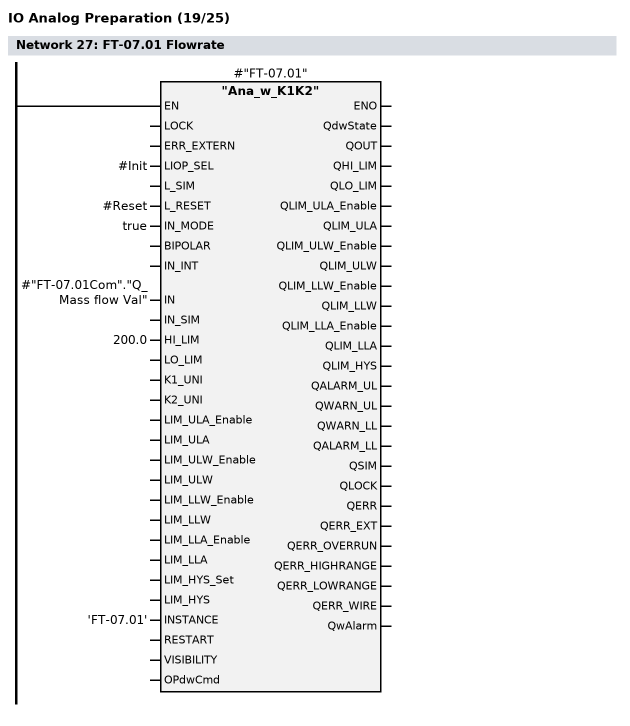
   RUNG wire#powerrail
      #"FT-07.01"(LOCK :=, ERR_EXTERN :=, LIOP_SEL := #Init, L_SIM :=, L_RESET := #Reset, IN_MODE := true, BIPOLAR :=, IN_INT :=, IN := #"FT-07.01Com"."Q_Mass flow Val", IN_SIM :=, HI_LIM := 200.0, LO_LIM :=, K1_UNI :=, K2_UNI :=, LIM_ULA_Enable :=, LIM_ULA :=, LIM_ULW_Enable :=, LIM_ULW :=, LIM_LLW_Enable :=, LIM_LLW :=, LIM_LLA_Enable :=, LIM_LLA :=, LIM_HYS_Set :=, LIM_HYS :=, INSTANCE := 'FT-07.01', RESTART :=, VISIBILITY :=, OPdwCmd :=, QdwState =>, QOUT =>, QHI_LIM =>, QLO_LIM =>, QLIM_ULA_Enable =>, QLIM_ULA =>, QLIM_ULW_Enable =>, QLIM_ULW =>, QLIM_LLW_Enable =>, QLIM_LLW =>, QLIM_LLA_Enable =>, QLIM_LLA =>, QLIM_HYS =>, QALARM_UL =>, QWARN_UL =>, QWARN_LL =>, QALARM_LL =>, QSIM =>, QLOCK =>, QERR =>, QERR_EXT =>, QERR_OVERRUN =>, QERR_HIGHRANGE =>, QERR_LOWRANGE =>, QERR_WIRE =>, QwAlarm =>)
   END_RUNG
   // the same network as SCL:
   #"FT-07.01"(LIOP_SEL := #Init,   // "Ana_w_K1K2"
               L_RESET := #Reset,
               IN_MODE := true,
               IN := #"FT-07.01Com"."Q_Mass flow Val",
               HI_LIM := 200.0,
               INSTANCE := 'FT-07.01');
END_REGION

REGION Network 28: FT-08.01 Communication
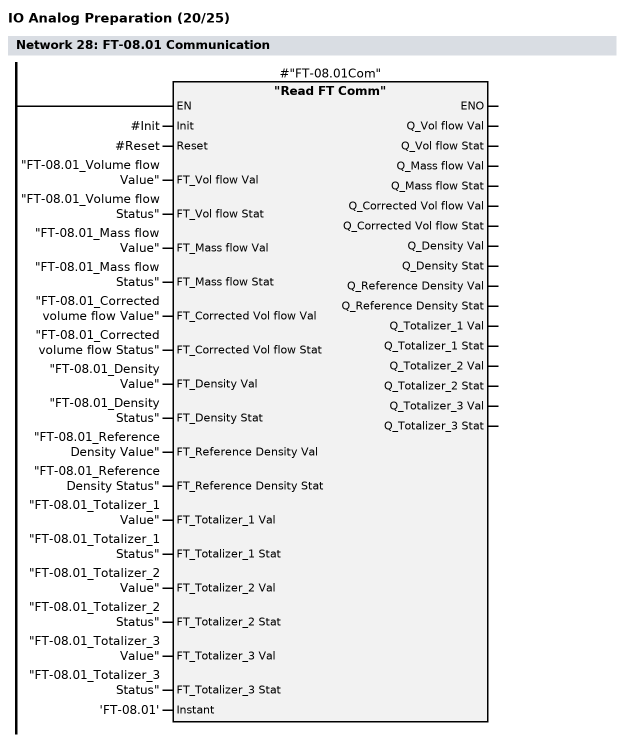
   RUNG wire#powerrail
      #"FT-08.01Com"(Init := #Init, Reset := #Reset, "FT_Vol flow Val" := "FT-08.01_Volume flow Value", "FT_Vol flow Stat" := "FT-08.01_Volume flow Status", "FT_Mass flow Val" := "FT-08.01_Mass flow Value", "FT_Mass flow Stat" := "FT-08.01_Mass flow Status", "FT_Corrected Vol flow Val" := "FT-08.01_Corrected volume flow Value", "FT_Corrected Vol flow Stat" := "FT-08.01_Corrected volume flow Status", "FT_Density Val" := "FT-08.01_Density Value", "FT_Density Stat" := "FT-08.01_Density Status", "FT_Reference Density Val" := "FT-08.01_Reference Density Value", "FT_Reference Density Stat" := "FT-08.01_Reference Density Status", "FT_Totalizer_1 Val" := "FT-08.01_Totalizer_1 Value", "FT_Totalizer_1 Stat" := "FT-08.01_Totalizer_1 Status", "FT_Totalizer_2 Val" := "FT-08.01_Totalizer_2 Value", "FT_Totalizer_2 Stat" := "FT-08.01_Totalizer_2 Status", "FT_Totalizer_3 Val" := "FT-08.01_Totalizer_3 Value", "FT_Totalizer_3 Stat" := "FT-08.01_Totalizer_3 Status", Instant := 'FT-08.01', "Q_Vol flow Val" =>, "Q_Vol flow Stat" =>, "Q_Mass flow Val" =>, "Q_Mass flow Stat" =>, "Q_Corrected Vol flow Val" =>, "Q_Corrected Vol flow Stat" =>, "Q_Density Val" =>, "Q_Density Stat" =>, "Q_Reference Density Val" =>, "Q_Reference Density Stat" =>, "Q_Totalizer_1 Val" =>, "Q_Totalizer_1 Stat" =>, "Q_Totalizer_2 Val" =>, "Q_Totalizer_2 Stat" =>, "Q_Totalizer_3 Val" =>, "Q_Totalizer_3 Stat" =>)
   END_RUNG
   // the same network as SCL:
   #"FT-08.01Com"(Init := #Init,   // "Read FT Comm"
                  Reset := #Reset,
                  "FT_Vol flow Val" := "FT-08.01_Volume flow Value",
                  "FT_Vol flow Stat" := "FT-08.01_Volume flow Status",
                  "FT_Mass flow Val" := "FT-08.01_Mass flow Value",
                  "FT_Mass flow Stat" := "FT-08.01_Mass flow Status",
                  "FT_Corrected Vol flow Val" := "FT-08.01_Corrected volume flow Value",
                  "FT_Corrected Vol flow Stat" := "FT-08.01_Corrected volume flow Status",
                  "FT_Density Val" := "FT-08.01_Density Value",
                  "FT_Density Stat" := "FT-08.01_Density Status",
                  "FT_Reference Density Val" := "FT-08.01_Reference Density Value",
                  "FT_Reference Density Stat" := "FT-08.01_Reference Density Status",
                  "FT_Totalizer_1 Val" := "FT-08.01_Totalizer_1 Value",
                  "FT_Totalizer_1 Stat" := "FT-08.01_Totalizer_1 Status",
                  "FT_Totalizer_2 Val" := "FT-08.01_Totalizer_2 Value",
                  "FT_Totalizer_2 Stat" := "FT-08.01_Totalizer_2 Status",
                  "FT_Totalizer_3 Val" := "FT-08.01_Totalizer_3 Value",
                  "FT_Totalizer_3 Stat" := "FT-08.01_Totalizer_3 Status",
                  Instant := 'FT-08.01');
END_REGION

REGION Network 29: FT-08.01 Flowrate
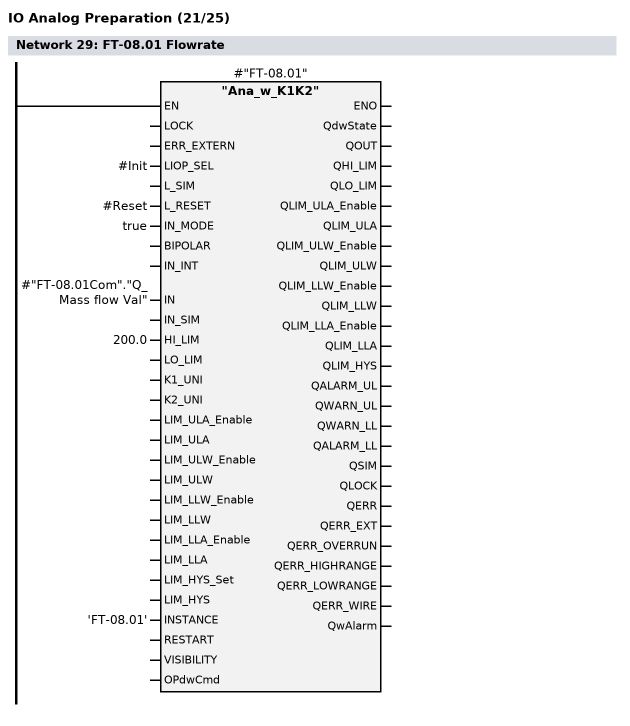
   RUNG wire#powerrail
      #"FT-08.01"(LOCK :=, ERR_EXTERN :=, LIOP_SEL := #Init, L_SIM :=, L_RESET := #Reset, IN_MODE := true, BIPOLAR :=, IN_INT :=, IN := #"FT-08.01Com"."Q_Mass flow Val", IN_SIM :=, HI_LIM := 200.0, LO_LIM :=, K1_UNI :=, K2_UNI :=, LIM_ULA_Enable :=, LIM_ULA :=, LIM_ULW_Enable :=, LIM_ULW :=, LIM_LLW_Enable :=, LIM_LLW :=, LIM_LLA_Enable :=, LIM_LLA :=, LIM_HYS_Set :=, LIM_HYS :=, INSTANCE := 'FT-08.01', RESTART :=, VISIBILITY :=, OPdwCmd :=, QdwState =>, QOUT =>, QHI_LIM =>, QLO_LIM =>, QLIM_ULA_Enable =>, QLIM_ULA =>, QLIM_ULW_Enable =>, QLIM_ULW =>, QLIM_LLW_Enable =>, QLIM_LLW =>, QLIM_LLA_Enable =>, QLIM_LLA =>, QLIM_HYS =>, QALARM_UL =>, QWARN_UL =>, QWARN_LL =>, QALARM_LL =>, QSIM =>, QLOCK =>, QERR =>, QERR_EXT =>, QERR_OVERRUN =>, QERR_HIGHRANGE =>, QERR_LOWRANGE =>, QERR_WIRE =>, QwAlarm =>)
   END_RUNG
   // the same network as SCL:
   #"FT-08.01"(LIOP_SEL := #Init,   // "Ana_w_K1K2"
               L_RESET := #Reset,
               IN_MODE := true,
               IN := #"FT-08.01Com"."Q_Mass flow Val",
               HI_LIM := 200.0,
               INSTANCE := 'FT-08.01');
END_REGION

REGION Network 30: FT-09.01 Communication
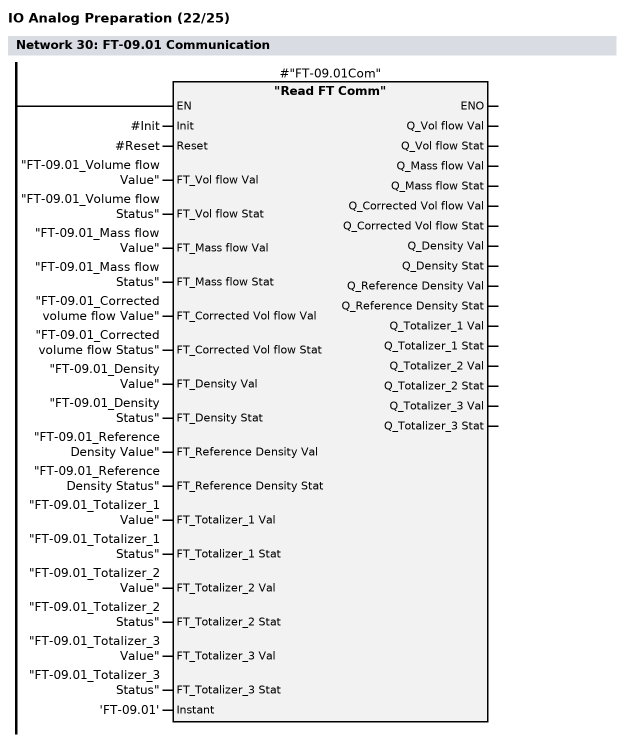
   RUNG wire#powerrail
      #"FT-09.01Com"(Init := #Init, Reset := #Reset, "FT_Vol flow Val" := "FT-09.01_Volume flow Value", "FT_Vol flow Stat" := "FT-09.01_Volume flow Status", "FT_Mass flow Val" := "FT-09.01_Mass flow Value", "FT_Mass flow Stat" := "FT-09.01_Mass flow Status", "FT_Corrected Vol flow Val" := "FT-09.01_Corrected volume flow Value", "FT_Corrected Vol flow Stat" := "FT-09.01_Corrected volume flow Status", "FT_Density Val" := "FT-09.01_Density Value", "FT_Density Stat" := "FT-09.01_Density Status", "FT_Reference Density Val" := "FT-09.01_Reference Density Value", "FT_Reference Density Stat" := "FT-09.01_Reference Density Status", "FT_Totalizer_1 Val" := "FT-09.01_Totalizer_1 Value", "FT_Totalizer_1 Stat" := "FT-09.01_Totalizer_1 Status", "FT_Totalizer_2 Val" := "FT-09.01_Totalizer_2 Value", "FT_Totalizer_2 Stat" := "FT-09.01_Totalizer_2 Status", "FT_Totalizer_3 Val" := "FT-09.01_Totalizer_3 Value", "FT_Totalizer_3 Stat" := "FT-09.01_Totalizer_3 Status", Instant := 'FT-09.01', "Q_Vol flow Val" =>, "Q_Vol flow Stat" =>, "Q_Mass flow Val" =>, "Q_Mass flow Stat" =>, "Q_Corrected Vol flow Val" =>, "Q_Corrected Vol flow Stat" =>, "Q_Density Val" =>, "Q_Density Stat" =>, "Q_Reference Density Val" =>, "Q_Reference Density Stat" =>, "Q_Totalizer_1 Val" =>, "Q_Totalizer_1 Stat" =>, "Q_Totalizer_2 Val" =>, "Q_Totalizer_2 Stat" =>, "Q_Totalizer_3 Val" =>, "Q_Totalizer_3 Stat" =>)
   END_RUNG
   // the same network as SCL:
   #"FT-09.01Com"(Init := #Init,   // "Read FT Comm"
                  Reset := #Reset,
                  "FT_Vol flow Val" := "FT-09.01_Volume flow Value",
                  "FT_Vol flow Stat" := "FT-09.01_Volume flow Status",
                  "FT_Mass flow Val" := "FT-09.01_Mass flow Value",
                  "FT_Mass flow Stat" := "FT-09.01_Mass flow Status",
                  "FT_Corrected Vol flow Val" := "FT-09.01_Corrected volume flow Value",
                  "FT_Corrected Vol flow Stat" := "FT-09.01_Corrected volume flow Status",
                  "FT_Density Val" := "FT-09.01_Density Value",
                  "FT_Density Stat" := "FT-09.01_Density Status",
                  "FT_Reference Density Val" := "FT-09.01_Reference Density Value",
                  "FT_Reference Density Stat" := "FT-09.01_Reference Density Status",
                  "FT_Totalizer_1 Val" := "FT-09.01_Totalizer_1 Value",
                  "FT_Totalizer_1 Stat" := "FT-09.01_Totalizer_1 Status",
                  "FT_Totalizer_2 Val" := "FT-09.01_Totalizer_2 Value",
                  "FT_Totalizer_2 Stat" := "FT-09.01_Totalizer_2 Status",
                  "FT_Totalizer_3 Val" := "FT-09.01_Totalizer_3 Value",
                  "FT_Totalizer_3 Stat" := "FT-09.01_Totalizer_3 Status",
                  Instant := 'FT-09.01');
END_REGION

REGION Network 31: FT-09.01 Flowrate
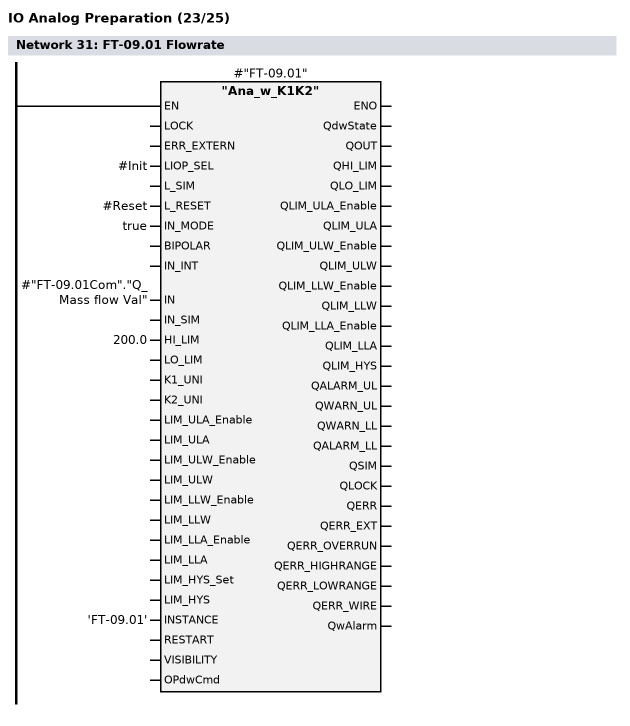
   RUNG wire#powerrail
      #"FT-09.01"(LOCK :=, ERR_EXTERN :=, LIOP_SEL := #Init, L_SIM :=, L_RESET := #Reset, IN_MODE := true, BIPOLAR :=, IN_INT :=, IN := #"FT-09.01Com"."Q_Mass flow Val", IN_SIM :=, HI_LIM := 200.0, LO_LIM :=, K1_UNI :=, K2_UNI :=, LIM_ULA_Enable :=, LIM_ULA :=, LIM_ULW_Enable :=, LIM_ULW :=, LIM_LLW_Enable :=, LIM_LLW :=, LIM_LLA_Enable :=, LIM_LLA :=, LIM_HYS_Set :=, LIM_HYS :=, INSTANCE := 'FT-09.01', RESTART :=, VISIBILITY :=, OPdwCmd :=, QdwState =>, QOUT =>, QHI_LIM =>, QLO_LIM =>, QLIM_ULA_Enable =>, QLIM_ULA =>, QLIM_ULW_Enable =>, QLIM_ULW =>, QLIM_LLW_Enable =>, QLIM_LLW =>, QLIM_LLA_Enable =>, QLIM_LLA =>, QLIM_HYS =>, QALARM_UL =>, QWARN_UL =>, QWARN_LL =>, QALARM_LL =>, QSIM =>, QLOCK =>, QERR =>, QERR_EXT =>, QERR_OVERRUN =>, QERR_HIGHRANGE =>, QERR_LOWRANGE =>, QERR_WIRE =>, QwAlarm =>)
   END_RUNG
   // the same network as SCL:
   #"FT-09.01"(LIOP_SEL := #Init,   // "Ana_w_K1K2"
               L_RESET := #Reset,
               IN_MODE := true,
               IN := #"FT-09.01Com"."Q_Mass flow Val",
               HI_LIM := 200.0,
               INSTANCE := 'FT-09.01');
END_REGION

REGION Network 32: FT-10.01 Communication
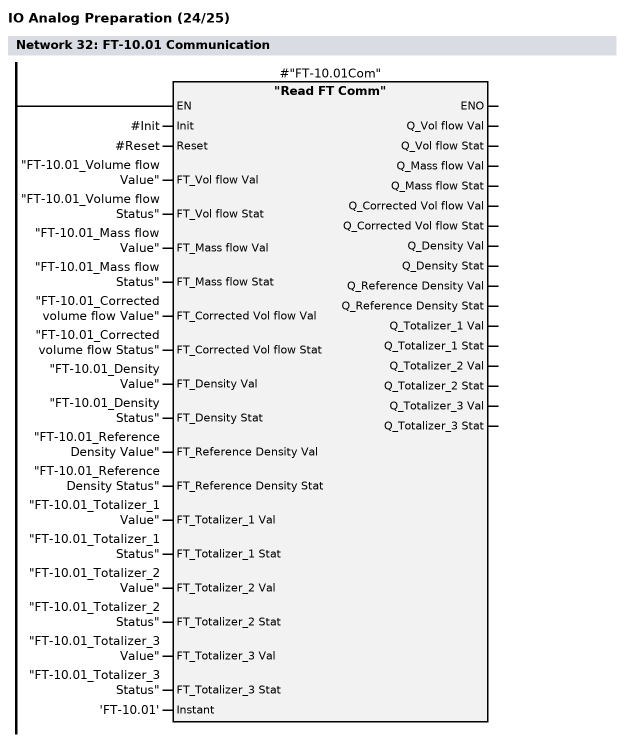
   RUNG wire#powerrail
      #"FT-10.01Com"(Init := #Init, Reset := #Reset, "FT_Vol flow Val" := "FT-10.01_Volume flow Value", "FT_Vol flow Stat" := "FT-10.01_Volume flow Status", "FT_Mass flow Val" := "FT-10.01_Mass flow Value", "FT_Mass flow Stat" := "FT-10.01_Mass flow Status", "FT_Corrected Vol flow Val" := "FT-10.01_Corrected volume flow Value", "FT_Corrected Vol flow Stat" := "FT-10.01_Corrected volume flow Status", "FT_Density Val" := "FT-10.01_Density Value", "FT_Density Stat" := "FT-10.01_Density Status", "FT_Reference Density Val" := "FT-10.01_Reference Density Value", "FT_Reference Density Stat" := "FT-10.01_Reference Density Status", "FT_Totalizer_1 Val" := "FT-10.01_Totalizer_1 Value", "FT_Totalizer_1 Stat" := "FT-10.01_Totalizer_1 Status", "FT_Totalizer_2 Val" := "FT-10.01_Totalizer_2 Value", "FT_Totalizer_2 Stat" := "FT-10.01_Totalizer_2 Status", "FT_Totalizer_3 Val" := "FT-10.01_Totalizer_3 Value", "FT_Totalizer_3 Stat" := "FT-10.01_Totalizer_3 Status", Instant := 'FT-10.01', "Q_Vol flow Val" =>, "Q_Vol flow Stat" =>, "Q_Mass flow Val" =>, "Q_Mass flow Stat" =>, "Q_Corrected Vol flow Val" =>, "Q_Corrected Vol flow Stat" =>, "Q_Density Val" =>, "Q_Density Stat" =>, "Q_Reference Density Val" =>, "Q_Reference Density Stat" =>, "Q_Totalizer_1 Val" =>, "Q_Totalizer_1 Stat" =>, "Q_Totalizer_2 Val" =>, "Q_Totalizer_2 Stat" =>, "Q_Totalizer_3 Val" =>, "Q_Totalizer_3 Stat" =>)
   END_RUNG
   // the same network as SCL:
   #"FT-10.01Com"(Init := #Init,   // "Read FT Comm"
                  Reset := #Reset,
                  "FT_Vol flow Val" := "FT-10.01_Volume flow Value",
                  "FT_Vol flow Stat" := "FT-10.01_Volume flow Status",
                  "FT_Mass flow Val" := "FT-10.01_Mass flow Value",
                  "FT_Mass flow Stat" := "FT-10.01_Mass flow Status",
                  "FT_Corrected Vol flow Val" := "FT-10.01_Corrected volume flow Value",
                  "FT_Corrected Vol flow Stat" := "FT-10.01_Corrected volume flow Status",
                  "FT_Density Val" := "FT-10.01_Density Value",
                  "FT_Density Stat" := "FT-10.01_Density Status",
                  "FT_Reference Density Val" := "FT-10.01_Reference Density Value",
                  "FT_Reference Density Stat" := "FT-10.01_Reference Density Status",
                  "FT_Totalizer_1 Val" := "FT-10.01_Totalizer_1 Value",
                  "FT_Totalizer_1 Stat" := "FT-10.01_Totalizer_1 Status",
                  "FT_Totalizer_2 Val" := "FT-10.01_Totalizer_2 Value",
                  "FT_Totalizer_2 Stat" := "FT-10.01_Totalizer_2 Status",
                  "FT_Totalizer_3 Val" := "FT-10.01_Totalizer_3 Value",
                  "FT_Totalizer_3 Stat" := "FT-10.01_Totalizer_3 Status",
                  Instant := 'FT-10.01');
END_REGION

REGION Network 33: FT-10.01 Flowrate
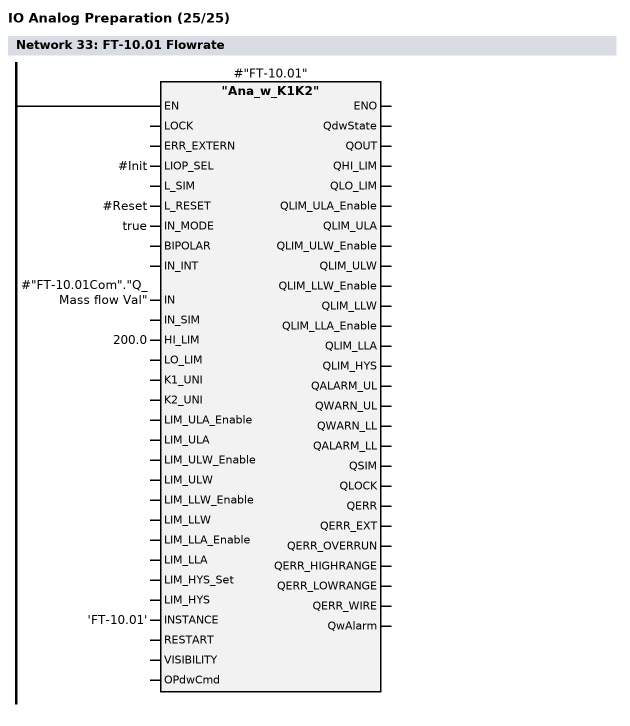
   RUNG wire#powerrail
      #"FT-10.01"(LOCK :=, ERR_EXTERN :=, LIOP_SEL := #Init, L_SIM :=, L_RESET := #Reset, IN_MODE := true, BIPOLAR :=, IN_INT :=, IN := #"FT-10.01Com"."Q_Mass flow Val", IN_SIM :=, HI_LIM := 200.0, LO_LIM :=, K1_UNI :=, K2_UNI :=, LIM_ULA_Enable :=, LIM_ULA :=, LIM_ULW_Enable :=, LIM_ULW :=, LIM_LLW_Enable :=, LIM_LLW :=, LIM_LLA_Enable :=, LIM_LLA :=, LIM_HYS_Set :=, LIM_HYS :=, INSTANCE := 'FT-10.01', RESTART :=, VISIBILITY :=, OPdwCmd :=, QdwState =>, QOUT =>, QHI_LIM =>, QLO_LIM =>, QLIM_ULA_Enable =>, QLIM_ULA =>, QLIM_ULW_Enable =>, QLIM_ULW =>, QLIM_LLW_Enable =>, QLIM_LLW =>, QLIM_LLA_Enable =>, QLIM_LLA =>, QLIM_HYS =>, QALARM_UL =>, QWARN_UL =>, QWARN_LL =>, QALARM_LL =>, QSIM =>, QLOCK =>, QERR =>, QERR_EXT =>, QERR_OVERRUN =>, QERR_HIGHRANGE =>, QERR_LOWRANGE =>, QERR_WIRE =>, QwAlarm =>)
   END_RUNG
   // the same network as SCL:
   #"FT-10.01"(LIOP_SEL := #Init,   // "Ana_w_K1K2"
               L_RESET := #Reset,
               IN_MODE := true,
               IN := #"FT-10.01Com"."Q_Mass flow Val",
               HI_LIM := 200.0,
               INSTANCE := 'FT-10.01');
END_REGION
END_FUNCTION_BLOCK

FUNCTION_BLOCK "Ana_w_K1K2"
TITLE = Analogue
{ S7_Optimized_Access := 'FALSE' }
AUTHOR : RM
FAMILY : MON
VERSION : 0.1
   VAR_INPUT 
      LOCK : Bool;
      ERR_EXTERN : Bool;
      LIOP_SEL : Bool;
      L_SIM : Bool;
      L_RESET : Bool;
      IN_MODE : Bool;
      BIPOLAR : Bool;
      IN_INT : Int := 0;
      IN : Real := 55.0;
      IN_SIM : Real := 55.0;
      HI_LIM : Real := 100.0;
      LO_LIM : Real;
      K1_UNI : Real;   // Low Measuring Unit
      K2_UNI : Real := 27648.0;   // High Mesuring Unit
      LIM_ULA_Enable : Bool;
      LIM_ULA : Real := 90.0;
      LIM_ULW_Enable : Bool;
      LIM_ULW : Real := 80.0;
      LIM_LLW_Enable : Bool;
      LIM_LLW : Real := 20.0;
      LIM_LLA_Enable : Bool;
      LIM_LLA : Real := 10.0;
      LIM_HYS_Set : Bool;
      LIM_HYS : Real;
      INSTANCE : String := 'Analogue_001';
      RESTART : Bool;
   END_VAR

   VAR_OUTPUT 
      QdwState : DWord;
      QOUT : Real;
      QHI_LIM : Real;
      QLO_LIM : Real;
      QLIM_ULA_Enable : Bool;
      QLIM_ULA : Real;
      QLIM_ULW_Enable : Bool;
      QLIM_ULW : Real;
      QLIM_LLW_Enable : Bool;
      QLIM_LLW : Real;
      QLIM_LLA_Enable : Bool;
      QLIM_LLA : Real;
      QLIM_HYS : Real;
      QALARM_UL : Bool;
      QWARN_UL : Bool;
      QWARN_LL : Bool;
      QALARM_LL : Bool;
      QSIM : Bool;
      QLOCK : Bool;
      QERR : Bool;
      QERR_EXT : Bool;
      QERR_OVERRUN : Bool;
      QERR_HIGHRANGE : Bool;
      QERR_LOWRANGE : Bool;
      QERR_WIRE : Bool;
      QwAlarm : Word;
   END_VAR

   VAR_IN_OUT 
      VISIBILITY : Byte := 0;
      OPdwCmd : DWord;
   END_VAR

   VAR 
      OP_RESET : Bool;
      QLIM_HYS_Set : Bool;
      QIN_MODE : Bool;
      OP_LIM_ULA : Real;
      OP_LIM_ULW : Real;
      OP_LIM_LLW : Real;
      OP_LIM_LLA : Real;
      OP_SIM_Value : Real;
      OP_LIM_HYS_Perc : Real;
      OP_LIM_HYS_Abs : Real;
      OP_HI_LIM : Real;
      OP_LO_LIM : Real;
      OP_VISIBILITY : Byte;
      VISIBILITY_OLD : Byte;
      SEF_L_RESET_Link : Bool;
      Condition_SEF_L_RESET_Link : Bool;
      SEF_L_RESET_OP : Bool;
      Condition_Enable_ULA : Bool;
      Condition_Enable_ULW : Bool;
      Condition_Enable_LLW : Bool;
      Condition_Enable_LLA : Bool;
   END_VAR


BEGIN
	(*
	Network 1: Start up
	*)
	IF #RESTART= true THEN
	  #QOUT:= 0;
	  #OPdwCmd:=0;
	END_IF;
	
	(*
	Network 2: Simulation On/Off
	Vaiable: OPdwCmd  Bit:  20  =  Process
	Vaiable: OPdwCmd  Bit:  21  =  Simulation
	*)
	IF (#LIOP_SEL=true AND #L_SIM=true) OR (#OPdwCmd.%X21=true AND #LIOP_SEL=false) THEN
	  #QSIM:=true;
	  #OPdwCmd.%X20:=false;
	  #OPdwCmd.%X21:=false;
	ELSIF (#LIOP_SEL=true AND #L_SIM=false) OR (#OPdwCmd.%X20=true AND #LIOP_SEL=false) THEN
	  #QSIM:= false;
	  #OPdwCmd.%X20:=false;
	  #OPdwCmd.%X21:=false;
	END_IF;
	
	(*
	Network 3: Mode limit Hysteresis
	Vaiable: OPdwCmd  Bit:  12  =  Hysteresis Percental
	Vaiable: OPdwCmd  Bit:  13  =  Hysteresis Absolute
	*)
	IF (#LIOP_SEL=true AND #LIM_HYS_Set=true) OR (#OPdwCmd.%X13=true AND #LIOP_SEL=false) THEN
	  #QLIM_HYS_Set:=true;
	  #OPdwCmd.%X12:=false;
	  #OPdwCmd.%X13:=false;
	ELSIF (#LIOP_SEL=true AND #LIM_HYS_Set=false) OR (#OPdwCmd.%X12=true AND #LIOP_SEL=false) THEN
	  #QLIM_HYS_Set:=false;
	  #OPdwCmd.%X12:=false;
	  #OPdwCmd.%X13:=false;
	END_IF;
	
	(*
	Network 4: Mode Periphery / Real value
	Vaiable: OPdwCmd  Bit:  14  =  Periphery
	Vaiable: OPdwCmd  Bit:  15  =  Real value
	*)
	IF (#LIOP_SEL=true AND #IN_MODE=true) OR (#OPdwCmd.%X15=true AND #LIOP_SEL=false) THEN
	  #QIN_MODE:=true;
	  #OPdwCmd.%X14:=false;
	  #OPdwCmd.%X15:=false;
	ELSIF (#LIOP_SEL=true AND #IN_MODE=false) OR (#OPdwCmd.%X14=true AND #LIOP_SEL=false) THEN
	  #QIN_MODE:=false;
	  #OPdwCmd.%X14:=false;
	  #OPdwCmd.%X15:=false;
	END_IF;
	
	(*
	Network 5: Reset Operation
	Vaiable: OPdwCmd  Bit:  24  =  Reset
	*)
	// Rising edge by linking
	IF #L_RESET=true AND #Condition_SEF_L_RESET_Link=false THEN
	  #SEF_L_RESET_Link:=true;
	  #Condition_SEF_L_RESET_Link:=true;
	ELSIF #L_RESET=true AND #Condition_SEF_L_RESET_Link=true THEN
	  #SEF_L_RESET_Link:=false;
	ELSE
	  #Condition_SEF_L_RESET_Link:=false;
	END_IF;
	// Rising edge by operator
	IF #OPdwCmd.%X24=true THEN
	  #SEF_L_RESET_OP:=true;
	  #OPdwCmd.%X24:=false;
	ELSE
	  #SEF_L_RESET_OP:=false;
	END_IF;
	// Reset error #OP_RESET:=(#LIOP_SEL=true AND #SEF_L_RESET_Link=true) OR (#SEF_L_RESET_OP=true AND #LIOP_SEL=false);
	#OP_RESET:=(#L_RESET=true) OR (#SEF_L_RESET_OP=true AND #LIOP_SEL=false);
	
	(*
	Network 6: Enable alarm for upper limit
	Vaiable: OPdwCmd  Bit:  0  =  Enable alarm upper limit
	*)
	IF #OPdwCmd.%X0=true THEN
	  #Condition_Enable_ULA:=NOT #Condition_Enable_ULA;
	  #OPdwCmd.%X0:=false;
	END_IF;
	//IF (#LIOP_SEL=true AND #LIM_ULA_Enable=true) OR (#LIOP_SEL=false AND #Condition_Enable_ULA=true) THEN  
	//#QLIM_ULA_Enable := true;
	//ELSIF (#LIOP_SEL=true AND #LIM_ULA_Enable=false) OR (#LIOP_SEL=false AND #Condition_Enable_ULA=false) THEN
	//    #QLIM_ULA_Enable := false;
	//END_IF;
	IF ( #LIM_ULA_Enable=true) OR (#LIOP_SEL=false AND #Condition_Enable_ULA=true) THEN  
	  #QLIM_ULA_Enable:=true;
	ELSIF (#LIOP_SEL=true AND #LIM_ULA_Enable=false) OR (#LIOP_SEL=false AND #Condition_Enable_ULA=false) THEN
	  #QLIM_ULA_Enable:=false;
	END_IF;
	
	  
	(*
	Network 7: Enable warning for upper limit
	Vaiable: OPdwCmd  Bit:  1  =  Enable warning upper limit
	*)
	IF #OPdwCmd.%X1=true THEN
	  #Condition_Enable_ULW:=NOT #Condition_Enable_ULW;
	  #OPdwCmd.%X1:=false;
	END_IF;
	
	IF ( #LIM_ULW_Enable=true) OR (#LIOP_SEL=false AND #Condition_Enable_ULW=true) THEN  
	  #QLIM_ULW_Enable:=true;
	ELSIF (#LIOP_SEL=true AND #LIM_ULW_Enable=false) OR (#LIOP_SEL=false AND #Condition_Enable_ULW=false) THEN
	  #QLIM_ULW_Enable:=false;
	END_IF;
	
	(*
	Network 8: Enable warning for lower limit
	Vaiable: OPdwCmd  Bit:  2  =  Enable warning lower limit
	*)
	IF #OPdwCmd.%X2=true THEN
	  #Condition_Enable_LLW:=NOT #Condition_Enable_LLW ;
	  #OPdwCmd.%X2:=false;
	END_IF;
	
	IF ( #LIM_LLW_Enable=true) OR (#LIOP_SEL=false AND #Condition_Enable_LLW=true) THEN  
	  #QLIM_LLW_Enable:=true;
	ELSIF (#LIOP_SEL=true AND #LIM_LLW_Enable=false) OR (#LIOP_SEL=false AND #Condition_Enable_LLW=false) THEN
	  #QLIM_LLW_Enable:=false;
	END_IF;
	
	(*
	Network 9: Enable alarm for lower limit
	Vaiable: OPdwCmd  Bit:  3  =  Enable alarm lower limit
	*)
	IF #OPdwCmd.%X3=true THEN
	  #Condition_Enable_LLA:=NOT #Condition_Enable_LLA;
	  #OPdwCmd.%X3:=false;
	END_IF;
	
	IF ( #LIM_LLA_Enable=true) OR (#LIOP_SEL=false AND #Condition_Enable_LLA=true) THEN  
	  #QLIM_LLA_Enable:=true;
	ELSIF (#LIOP_SEL=true AND #LIM_LLA_Enable=false) OR (#LIOP_SEL=false AND #Condition_Enable_LLA=false) THEN
	  #QLIM_LLA_Enable:=false;
	END_IF;
	
	(*
	Network 10: Calculate hysteresis value
	*)
	IF #LIOP_SEL=true AND #QLIM_HYS_Set=true THEN
	  // Absolute by PLC
	  #OP_HI_LIM:=#HI_LIM;
	  #OP_LO_LIM:=#LO_LIM;
	  #OP_LIM_HYS_Perc:=#LIM_HYS/((#HI_LIM-#LO_LIM)/100);
	  #OP_LIM_HYS_Abs:=#LIM_HYS;
	  #QHI_LIM:=#HI_LIM;
	  #QLO_LIM:=#LO_LIM;
	  #QLIM_HYS:=#OP_LIM_HYS_Abs;
	ELSIF #LIOP_SEL=true AND #QLIM_HYS_Set=false THEN
	  // Percental by PLC
	  #OP_HI_LIM:=#HI_LIM;
	  #OP_LO_LIM:=#LO_LIM;
	  #OP_LIM_HYS_Perc:=#LIM_HYS;
	  #OP_LIM_HYS_Abs:=#LIM_HYS*((#HI_LIM-#LO_LIM)/100);
	  #QHI_LIM:=#HI_LIM;
	  #QLO_LIM:=#LO_LIM;
	  #QLIM_HYS:=#OP_LIM_HYS_Abs;
	ELSIF #LIOP_SEL=false AND #QLIM_HYS_Set=true THEN
	  // Absolute by operator
	  #QHI_LIM:=#OP_HI_LIM;
	  #QLO_LIM:=#OP_LO_LIM;
	  #OP_LIM_HYS_Perc:=#OP_LIM_HYS_Abs/((#OP_HI_LIM-#OP_LO_LIM)/100);
	  #QLIM_HYS:=#OP_LIM_HYS_Abs;
	ELSE
	  // Percental by operator
	  #QHI_LIM:=#OP_HI_LIM;
	  #QLO_LIM:=#OP_LO_LIM;
	  #OP_LIM_HYS_Abs:=#OP_LIM_HYS_Perc*((#OP_HI_LIM-#OP_LO_LIM)/100);
	  #QLIM_HYS:=#OP_LIM_HYS_Abs;
	END_IF;
	
	//Transfer output to simulation value in process mode
	IF #QSIM=false THEN
	  #IN_SIM:=#QOUT;
	END_IF;
	(*
	Network 11: Convert integer to real and scale it to selcted mode
	*)
	IF #QIN_MODE=false AND #QSIM=false AND #BIPOLAR=false THEN
	  // Convert integer to real and scale in unipolar mode (4..20mA)
	    #QOUT:=(((INT_TO_REAL(#IN_INT)-#K1_UNI)/#K2_UNI)*(#HI_LIM-#LO_LIM))+#LO_LIM;
	ELSIF #QIN_MODE=false AND #QSIM=false AND #BIPOLAR=true THEN
	  // Convert integer to real and scale in bipolar mode (4..20mA)
	  #QOUT:=(((INT_TO_REAL(#IN_INT)+27648)/55296)*(#HI_LIM-#LO_LIM))+#LO_LIM;
	END_IF;
	
	//Che errors
	#QERR_EXT:=#ERR_EXTERN;
	#QLOCK:=#LOCK;
	
	(*
	Network 12: Check errors for simulation mode or real value
	*)
	IF (#QIN_MODE=true OR #QSIM=true) AND #QHI_LIM>=#QOUT AND #QLO_LIM<=#QOUT THEN
	    #QERR_OVERRUN:=false;
	    #QERR_HIGHRANGE:=false;
	    #QERR_LOWRANGE:=false;
	    #QERR_WIRE:=false;
	  END_IF;
	
	(*
	Network 13: Check errors for periphery unipolar mode (4..20mA)
	*)
	(*
	    Measuring Range   Units       Range
	    (4..20mA)         (Dez)
	    ============================================
	    >22,81            >32511      Overrun
	    --------------------------------------------
	    22,81              32511
	      .                           High range
	    20,01              27649         
	    --------------------------------------------
	    20,00              27648 
	      .                           Nominal range
	     4,00                  0
	    --------------------------------------------
	     3,99                 -1
	      .                           Low range
	     1,185             -4864
	    --------------------------------------------
	    <1,185            <-4864      Wire breakage
	*)
	IF #QSIM=false AND #QIN_MODE=false AND #BIPOLAR=false THEN
	  CASE #IN_INT OF
	      -4864..-1 :      // Low range
	    #QERR_OVERRUN:=false;
	    #QERR_HIGHRANGE:=false;
	   // #QERR_LOWRANGE := true;
	    #QERR_WIRE:=false;
	    0.. 27648:       // Nominal range
	    #QERR_OVERRUN:=false;
	    #QERR_HIGHRANGE:=false;
	    #QERR_LOWRANGE:=false;
	    #QERR_WIRE:=false;
	    27649..32511:   // High range
	    #QERR_OVERRUN:=false;
	    #QERR_HIGHRANGE:=true;
	    #QERR_LOWRANGE := false;
	    #QERR_WIRE:=false;
	  ELSE
	    IF #IN_INT>32511 THEN
	      // Overrun
	      #QERR_OVERRUN:=true;
	      #QERR_HIGHRANGE:=false;
	      #QERR_LOWRANGE:=false;
	      #QERR_WIRE:=false;
	    ELSE
	      // Wire breakage
	      #QERR_OVERRUN:=false;
	      #QERR_HIGHRANGE:=false;
	      #QERR_LOWRANGE:=false;
	      #QERR_WIRE:=true;
	    END_IF;  
	  END_CASE;
	END_IF;
	
	(*
	Network 14: Check errors for periphery bipolar mode (4..20mA)
	*)
	(*
	    Measuring Range   Units       Range
	    (4..20mA)         (Dez)
	    ============================================
	    >22,81            >32511      Overrun
	    --------------------------------------------
	    22,81              32511
	      .                           High range
	    20,01              27649         
	    --------------------------------------------
	    20,00              27648 
	      .                           Nominal range
	     4,00             -27648
	    --------------------------------------------
	     3,99             -27649
	      .                           Low range
	     1,185            -32512
	    --------------------------------------------
	    <1,185           <-32512      Wire breakage
	*)
	IF #QSIM=false AND #QIN_MODE=false AND #BIPOLAR=true THEN
	  CASE #IN_INT OF
	    -32512..-27649:         // Low range
	    #QERR_OVERRUN:=false;
	    #QERR_HIGHRANGE:=false;
	    #QERR_LOWRANGE:=true;
	    #QERR_WIRE:=false;
	    -27648..27648:         // Nominal range
	    #QERR_OVERRUN:=false;
	    #QERR_HIGHRANGE:=false;
	    #QERR_LOWRANGE:=false;
	    #QERR_WIRE:=false;
	    27649..32511:         // High range
	    #QERR_OVERRUN:=false;
	    #QERR_HIGHRANGE:=true;
	    #QERR_LOWRANGE:=false;
	    #QERR_WIRE:=false;
	  ELSE
	    IF #IN_INT>32511 THEN
	      // Overrun
	      #QERR_OVERRUN:=true;
	      #QERR_HIGHRANGE:=false;
	      #QERR_LOWRANGE:=false;
	      #QERR_WIRE:=false;
	    ELSE
	      // Wire breakage
	      #QERR_OVERRUN:=false;
	      #QERR_HIGHRANGE:=false;
	      #QERR_LOWRANGE:=false;
	      #QERR_WIRE:=true;
	    END_IF;  
	  END_CASE;
	END_IF;
	
	(*
	Network 15: Check range error for real value
	*)
	//  Check for high range injury
	IF (#IN>#QHI_LIM AND #QIN_MODE=true AND #QSIM=false AND #LIOP_SEL=true) OR
	   (#IN_SIM>#QHI_LIM AND #QSIM=true AND #LIOP_SEL=true) OR
	   (#OP_SIM_Value>#QHI_LIM AND #QSIM=true AND #LIOP_SEL=false) THEN
	      #QERR_HIGHRANGE:=true;
	END_IF;
	//  Check for low range injury
	IF (#IN<#QLO_LIM AND #QIN_MODE=true AND #QSIM=false AND #LIOP_SEL=true) OR
	   (#IN_SIM<#QLO_LIM AND #QSIM=true AND #LIOP_SEL=true) OR
	   (#OP_SIM_Value<#QLO_LIM AND #QSIM=true AND #LIOP_SEL=false) THEN
	      #QERR_LOWRANGE:=true;
	END_IF;
	    
	(*
	Network 16: General Error
	*)
	IF #OP_RESET=true THEN
	  #QERR:=false;
	ELSIF #QERR_EXT=true OR #QLOCK=true OR #QERR_OVERRUN OR #QERR_WIRE THEN
	  #QERR:=true;
	END_IF;
	
	(*
	Network 17: Upper limit alarm
	*)
	IF #QLIM_ULA_Enable=true THEN
	  IF #QLIM_ULA<=#QOUT THEN
	    #QALARM_UL:=true;
	  ELSIF (#QLIM_ULA-#QLIM_HYS)>#QOUT THEN
	    #QALARM_UL:=false;
	  END_IF;
	ELSE
	  #QALARM_UL:=false;
	END_IF;
	 
	(*
	Network 18: Upper limit warning
	*)
	IF #QLIM_ULW_Enable=true THEN
	  IF #QLIM_ULW<=#QOUT THEN
	    #QWARN_UL:=true;
	  ELSIF (#QLIM_ULW-#QLIM_HYS)>#QOUT THEN
	    #QWARN_UL:=false;
	  END_IF;
	ELSE
	  #QWARN_UL:=false;
	END_IF;
	
	(*
	Network 19: Lower limit warning
	*)
	IF #QLIM_LLW_Enable=true THEN
	  IF #QLIM_LLW>=#QOUT THEN
	    #QWARN_LL:=true;
	  ELSIF (#QLIM_LLW+#QLIM_HYS)<#QOUT THEN
	    #QWARN_LL:=false;
	  END_IF;
	ELSE
	  #QWARN_LL:=false;
	END_IF;
	
	(*
	Network 20: Lower limit alarm
	*)
	IF #QLIM_LLA_Enable=true THEN
	  IF #QLIM_LLA>=#QOUT THEN
	    #QALARM_LL:=true;
	  ELSIF (#QLIM_LLA+#QLIM_HYS)<#QOUT THEN
	    #QALARM_LL:=false;
	  END_IF;
	ELSE
	  #QALARM_LL:=false;
	END_IF;
	
	(*
	Network 21: Set limit value
	*)
	IF #QSIM=true AND #LIOP_SEL=false THEN
	  // Set values in simulation mode by operator
	  #QHI_LIM:=#OP_HI_LIM;
	  #QLO_LIM:=#OP_LO_LIM;
	  #QLIM_ULA:=#OP_LIM_ULA;
	  #QLIM_ULW:=#OP_LIM_ULW;
	  #QLIM_LLW:=#OP_LIM_LLW;
	  #QLIM_LLA:=#OP_LIM_LLA;
	ELSE
	  // Set values in normal mode by linking
	  #OP_HI_LIM:=#HI_LIM;
	  #QHI_LIM:=#HI_LIM;
	  #OP_LO_LIM:=#LO_LIM;
	  #QLO_LIM:=#LO_LIM;
	  #OP_LIM_ULA:=#LIM_ULA;
	  #QLIM_ULA:=#LIM_ULA;
	  #OP_LIM_ULW:=#LIM_ULW;
	  #QLIM_ULW:=#LIM_ULW;
	  #OP_LIM_LLW:=#LIM_LLW;
	  #QLIM_LLW:=#LIM_LLW;
	  #OP_LIM_LLA:=#LIM_LLA;
	  #QLIM_LLA:=#LIM_LLA;
	END_IF;
	
	(*
	Network 22: Check settings and values
	*)
	IF #QSIM=false AND #QIN_MODE=true THEN
	  // Set settings in process mode by PLC (real value)
	  #QOUT:=#IN;
	ELSIF #QSIM=true AND #LIOP_SEL=false THEN
	  // Set settings in simulation mode by operator (real value)
	  #QOUT:=#OP_SIM_Value;
	ELSIF #QSIM=true AND #LIOP_SEL=true THEN
	  // Set settings in simulation mode by PLC (real value)
	  #QOUT:=#IN_SIM;
	END_IF;
	
	IF #QSIM=false AND #LIOP_SEL=true AND #IN_MODE=false THEN
	  //Set settings in process mode by PLC (periphery)
	  IF #QERR_EXT=true OR #QLOCK=true THEN
	  //Set value in case of error
	    #QOUT:=#QLO_LIM;
	ELSE
	  IF #QOUT>#QHI_LIM THEN
	    #QOUT:=#QHI_LIM;
	  ELSIF #QOUT<#LO_LIM THEN
	    #QOUT:=#QLO_LIM;
	  END_IF;
	END_IF;
	END_IF;
	(*
	Network 23: Infuence visibility of faceplate window
	*)
	IF #OP_VISIBILITY<>#VISIBILITY_OLD THEN
	  #VISIBILITY_OLD:=#OP_VISIBILITY;
	  #VISIBILITY:=#OP_VISIBILITY;
	ELSIF #VISIBILITY<>#VISIBILITY_OLD THEN
	  #VISIBILITY_OLD:=#VISIBILITY;
	  #OP_VISIBILITY:=#VISIBILITY;
	END_IF;
	
	(*
	Network 24: Transfer output to simulation value in process mode
	*)
	IF #QSIM=false THEN
	  #IN_SIM:=#QOUT;
	END_IF;
	
	(*
	Network 25: Check errors
	*)
	#QERR_EXT:=#ERR_EXTERN;
	#QLOCK:=#LOCK;
	
	(*
	Network 26: Set state for HMI
	*)
	#QdwState.%X0:= #QIN_MODE;
	#QdwState.%X1:=#QLIM_HYS_Set;
	#QdwState.%X2:=false;
	#QdwState.%X3:=false;
	#QdwState.%X4:=#QLIM_ULA_Enable;
	#QdwState.%X5:=#QLIM_ULW_Enable;
	#QdwState.%X6:=#QLIM_LLW_Enable;
	#QdwState.%X7:=#QLIM_LLA_Enable;
	#QdwState.%X9:=#QALARM_LL OR #QALARM_UL;
	#QdwState.%X8:=NOT #QdwState.%X9 AND (#QWARN_LL OR #QWARN_UL);
	#QdwState.%X10:=false;
	#QdwState.%X11:=false;
	#QdwState.%X12:=#QERR_LOWRANGE;
	#QdwState.%X13:=#QERR_HIGHRANGE;
	#QdwState.%X14:=#QERR_OVERRUN;
	#QdwState.%X15:=#QERR_WIRE;
	#QdwState.%X16:=false;
	#QdwState.%X17:=false;
	#QdwState.%X18:=#QSIM;
	#QdwState.%X19:=false;
	#QdwState.%X20:=false;
	#QdwState.%X21:=false;
	#QdwState.%X22:=false;
	#QdwState.%X23:=false;
	#QdwState.%X24:=#QERR;
	#QdwState.%X25:=#QERR_EXT;
	#QdwState.%X26:=#QLOCK;
	#QdwState.%X27:=#LOCK;
	#QdwState.%X28:=false;
	#QdwState.%X29:=false;
	#QdwState.%X30:=false;
	#QdwState.%X31:=false;
	
	(*
	Network 27: Bit alarm procedure
	*)
	#QwAlarm.%X0:=#QALARM_LL;
	#QwAlarm.%X1:=#QALARM_UL;
	#QwAlarm.%X2:=false;
	#QwAlarm.%X3:=false;
	#QwAlarm.%X4:=#QLOCK;
	#QwAlarm.%X5:=false;
	#QwAlarm.%X6:=#QERR_EXT;
	#QwAlarm.%X7:=#QERR;
	#QwAlarm.%X8:=#QWARN_LL;
	#QwAlarm.%X9:=#QWARN_UL;
	#QwAlarm.%X10:=false;
	#QwAlarm.%X11:=false;
	#QwAlarm.%X12:=#LOCK;
	#QwAlarm.%X13:=false;
	#QwAlarm.%X14:=false;
	#QwAlarm.%X15:=#QSIM;
	
END_FUNCTION_BLOCK

FUNCTION_BLOCK "Read FT Comm"   // FB642, LAD
{ S7_Optimized_Access := 'FALSE' }
VERSION : 0.1
// stored: AutoNumber false, IsIECCheckEnabled false, SetENOAutomatically false, UDAEnableTagReadback false
   VAR_INPUT
      Init : Bool;
      Reset : Bool;
      "FT_Vol flow Val" : Real;   // FT_Volume flow Value
      "FT_Vol flow Stat" : Byte;   // FT_Volume flow Status
      "FT_Mass flow Val" : Real;   // FT_Mass flow Value
      "FT_Mass flow Stat" : Byte;   // FT_Mass flow Status
      "FT_Corrected Vol flow Val" : Real;   // FT_Corrected volume flow Value
      "FT_Corrected Vol flow Stat" : Byte;   // FT_Corrected volume flow Status
      "FT_Density Val" : Real;   // FT_Velocity Value
      "FT_Density Stat" : Byte;   // FT_Velocity Status
      "FT_Reference Density Val" : Real;
      "FT_Reference Density Stat" : Byte;
      "FT_Totalizer_1 Val" : Real;   // FT_Totalizer_1 Value
      "FT_Totalizer_1 Stat" : Byte;   // FT_Totalizer_1 Status
      "FT_Totalizer_2 Val" : Real;   // FT_Totalizer_2 Value
      "FT_Totalizer_2 Stat" : Byte;   // FT_Totalizer_2 Status
      "FT_Totalizer_3 Val" : Real;   // FT_Totalizer_3 Value
      "FT_Totalizer_3 Stat" : Byte;   // FT_Totalizer_3 Status
      Instant { ExternalAccessible := 'False'; ExternalVisible := 'False'; ExternalWritable := 'False'} : String;
   END_VAR
   VAR_OUTPUT
      "Q_Vol flow Val" : Real;   // FT_Volume flow Value
      "Q_Vol flow Stat" : Word;   // FT_Volume flow Status
      "Q_Mass flow Val" : Real;   // FT_Mass flow Value
      "Q_Mass flow Stat" : Word;   // FT_Mass flow Status
      "Q_Corrected Vol flow Val" : Real;   // FT_Corrected volume flow Value
      "Q_Corrected Vol flow Stat" : Word;   // FT_Corrected volume flow Status
      "Q_Density Val" : Real;   // FT_Velocity Value
      "Q_Density Stat" : Word;   // FT_Velocity Status
      "Q_Reference Density Val" : Real;
      "Q_Reference Density Stat" : Word;
      "Q_Totalizer_1 Val" : Real;   // FT_Totalizer_1 Value
      "Q_Totalizer_1 Stat" : Word;   // FT_Totalizer_1 Status
      "Q_Totalizer_2 Val" : Real;   // FT_Totalizer_2 Value
      "Q_Totalizer_2 Stat" : Word;   // FT_Totalizer_2 Status
      "Q_Totalizer_3 Val" : Real;   // FT_Totalizer_3 Value
      "Q_Totalizer_3 Stat" : Word;   // FT_Totalizer_3 Status
   END_VAR
   VAR DB_SPECIFIC
      Always_On : Bool;
   END_VAR
BEGIN

REGION Network 1: Aways On
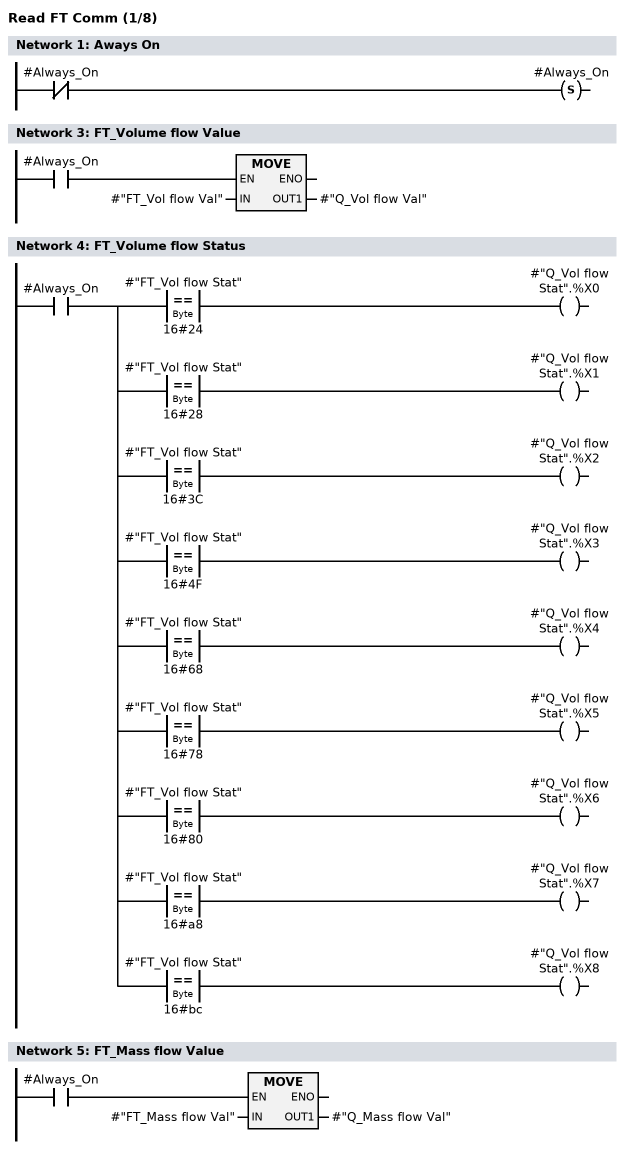
   RUNG wire#powerrail
      I_Contact( #Always_On )
      S_Coil( #Always_On )
   END_RUNG
   // the same network as SCL:
   IF NOT #Always_On THEN #Always_On := TRUE; END_IF;
END_REGION

REGION Network 2: Status Coding
   // 1. 0x24 : BAD - Maintenance alarm - A measured value is not available because a device error has occurred.
   // 2. 0x28 : BAD - Process related - A measured value is not available because the process
   // conditions are not within the device's technical specification limits.
   // 3. 0x3C : BAD - Function check - A function check is active (e.g. cleaning or calibration)
   // 4. 0x4F : UNCERTAIN - Initial value - A pre-defined value is output until a correct measured
   // value is available again or until remedial measures
   // have been carried out that change this status.
   // 5. 0x68 : UNCERTAIN - Maintenance demanded - Signs of wear and tear have been detected on the
   // measuring device. Short-term maintenance is needed to ensure that the measuring device remains
   // operational. The measured value might be invalid. The use of the measured value depends on the application.
   // 6. 0x78 : UNCERTAIN - Process related - The process conditions are not within the device's technical specification limits. This could have a negative impact on the quality and accuracy of the measured value. The use of the measured value depends on the application.
   // 7. 0x80 : GOOD - OK - No error has been diagnosed.
   // 8. 0xA8 : GOOD - Maintenance demanded -  The measured value is valid. It is highly advisable to service the device in the near future.
   // 9. 0xBC :  GOOD - Function check -  The measured value is valid. The measuring device is performing an internal function check. The function check does not have any noticeable effect on the process.
END_REGION

REGION Network 3: FT_Volume flow Value
   RUNG wire#powerrail
      Contact( #Always_On )
      Move(in := #"FT_Vol flow Val", out1 => #"Q_Vol flow Val")
   END_RUNG
   // the same network as SCL:
   IF #Always_On THEN #"Q_Vol flow Val" := #"FT_Vol flow Val"; END_IF;
END_REGION

REGION Network 4: FT_Volume flow Status
   RUNG wire#powerrail
      Contact( #Always_On )
      wire#w1
      { S7_Templates := "SrcType := Byte" } EQ_Contact(in1 := #"FT_Vol flow Stat", in2 := 16#24)
      Coil( #"Q_Vol flow Stat".%X0 )
   END_RUNG
   RUNG wire#w1
      { S7_Templates := "SrcType := Byte" } EQ_Contact(in1 := #"FT_Vol flow Stat", in2 := 16#28)
      Coil( #"Q_Vol flow Stat".%X1 )
   END_RUNG
   RUNG wire#w1
      { S7_Templates := "SrcType := Byte" } EQ_Contact(in1 := #"FT_Vol flow Stat", in2 := 16#3C)
      Coil( #"Q_Vol flow Stat".%X2 )
   END_RUNG
   RUNG wire#w1
      { S7_Templates := "SrcType := Byte" } EQ_Contact(in1 := #"FT_Vol flow Stat", in2 := 16#4F)
      Coil( #"Q_Vol flow Stat".%X3 )
   END_RUNG
   RUNG wire#w1
      { S7_Templates := "SrcType := Byte" } EQ_Contact(in1 := #"FT_Vol flow Stat", in2 := 16#68)
      Coil( #"Q_Vol flow Stat".%X4 )
   END_RUNG
   RUNG wire#w1
      { S7_Templates := "SrcType := Byte" } EQ_Contact(in1 := #"FT_Vol flow Stat", in2 := 16#78)
      Coil( #"Q_Vol flow Stat".%X5 )
   END_RUNG
   RUNG wire#w1
      { S7_Templates := "SrcType := Byte" } EQ_Contact(in1 := #"FT_Vol flow Stat", in2 := 16#80)
      Coil( #"Q_Vol flow Stat".%X6 )
   END_RUNG
   RUNG wire#w1
      { S7_Templates := "SrcType := Byte" } EQ_Contact(in1 := #"FT_Vol flow Stat", in2 := 16#a8)
      Coil( #"Q_Vol flow Stat".%X7 )
   END_RUNG
   RUNG wire#w1
      { S7_Templates := "SrcType := Byte" } EQ_Contact(in1 := #"FT_Vol flow Stat", in2 := 16#bc)
      Coil( #"Q_Vol flow Stat".%X8 )
   END_RUNG
   // the same network as SCL:
   #"Q_Vol flow Stat".%X0 := #Always_On AND (#"FT_Vol flow Stat" = 16#24);
   #"Q_Vol flow Stat".%X1 := #Always_On AND (#"FT_Vol flow Stat" = 16#28);
   #"Q_Vol flow Stat".%X2 := #Always_On AND (#"FT_Vol flow Stat" = 16#3C);
   #"Q_Vol flow Stat".%X3 := #Always_On AND (#"FT_Vol flow Stat" = 16#4F);
   #"Q_Vol flow Stat".%X4 := #Always_On AND (#"FT_Vol flow Stat" = 16#68);
   #"Q_Vol flow Stat".%X5 := #Always_On AND (#"FT_Vol flow Stat" = 16#78);
   #"Q_Vol flow Stat".%X6 := #Always_On AND (#"FT_Vol flow Stat" = 16#80);
   #"Q_Vol flow Stat".%X7 := #Always_On AND (#"FT_Vol flow Stat" = 16#a8);
   #"Q_Vol flow Stat".%X8 := #Always_On AND (#"FT_Vol flow Stat" = 16#bc);
END_REGION

REGION Network 5: FT_Mass flow Value
   RUNG wire#powerrail
      Contact( #Always_On )
      Move(in := #"FT_Mass flow Val", out1 => #"Q_Mass flow Val")
   END_RUNG
   // the same network as SCL:
   IF #Always_On THEN #"Q_Mass flow Val" := #"FT_Mass flow Val"; END_IF;
END_REGION

REGION Network 6: FT_Mass flow Status
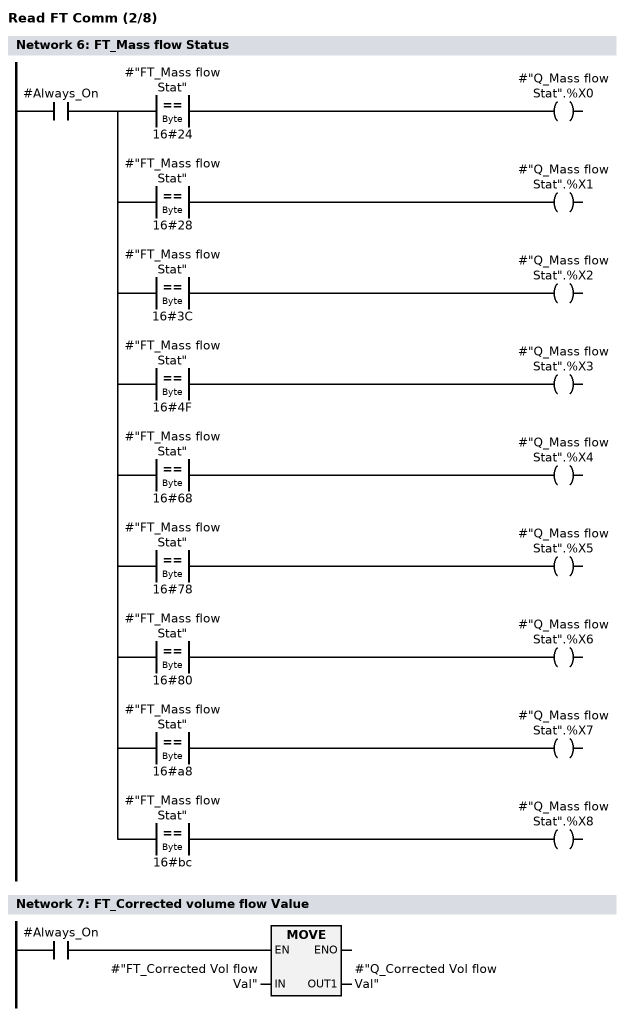
   RUNG wire#powerrail
      Contact( #Always_On )
      wire#w1
      { S7_Templates := "SrcType := Byte" } EQ_Contact(in1 := #"FT_Mass flow Stat", in2 := 16#24)
      Coil( #"Q_Mass flow Stat".%X0 )
   END_RUNG
   RUNG wire#w1
      { S7_Templates := "SrcType := Byte" } EQ_Contact(in1 := #"FT_Mass flow Stat", in2 := 16#28)
      Coil( #"Q_Mass flow Stat".%X1 )
   END_RUNG
   RUNG wire#w1
      { S7_Templates := "SrcType := Byte" } EQ_Contact(in1 := #"FT_Mass flow Stat", in2 := 16#3C)
      Coil( #"Q_Mass flow Stat".%X2 )
   END_RUNG
   RUNG wire#w1
      { S7_Templates := "SrcType := Byte" } EQ_Contact(in1 := #"FT_Mass flow Stat", in2 := 16#4F)
      Coil( #"Q_Mass flow Stat".%X3 )
   END_RUNG
   RUNG wire#w1
      { S7_Templates := "SrcType := Byte" } EQ_Contact(in1 := #"FT_Mass flow Stat", in2 := 16#68)
      Coil( #"Q_Mass flow Stat".%X4 )
   END_RUNG
   RUNG wire#w1
      { S7_Templates := "SrcType := Byte" } EQ_Contact(in1 := #"FT_Mass flow Stat", in2 := 16#78)
      Coil( #"Q_Mass flow Stat".%X5 )
   END_RUNG
   RUNG wire#w1
      { S7_Templates := "SrcType := Byte" } EQ_Contact(in1 := #"FT_Mass flow Stat", in2 := 16#80)
      Coil( #"Q_Mass flow Stat".%X6 )
   END_RUNG
   RUNG wire#w1
      { S7_Templates := "SrcType := Byte" } EQ_Contact(in1 := #"FT_Mass flow Stat", in2 := 16#a8)
      Coil( #"Q_Mass flow Stat".%X7 )
   END_RUNG
   RUNG wire#w1
      { S7_Templates := "SrcType := Byte" } EQ_Contact(in1 := #"FT_Mass flow Stat", in2 := 16#bc)
      Coil( #"Q_Mass flow Stat".%X8 )
   END_RUNG
   // the same network as SCL:
   #"Q_Mass flow Stat".%X0 := #Always_On AND (#"FT_Mass flow Stat" = 16#24);
   #"Q_Mass flow Stat".%X1 := #Always_On AND (#"FT_Mass flow Stat" = 16#28);
   #"Q_Mass flow Stat".%X2 := #Always_On AND (#"FT_Mass flow Stat" = 16#3C);
   #"Q_Mass flow Stat".%X3 := #Always_On AND (#"FT_Mass flow Stat" = 16#4F);
   #"Q_Mass flow Stat".%X4 := #Always_On AND (#"FT_Mass flow Stat" = 16#68);
   #"Q_Mass flow Stat".%X5 := #Always_On AND (#"FT_Mass flow Stat" = 16#78);
   #"Q_Mass flow Stat".%X6 := #Always_On AND (#"FT_Mass flow Stat" = 16#80);
   #"Q_Mass flow Stat".%X7 := #Always_On AND (#"FT_Mass flow Stat" = 16#a8);
   #"Q_Mass flow Stat".%X8 := #Always_On AND (#"FT_Mass flow Stat" = 16#bc);
END_REGION

REGION Network 7: FT_Corrected volume flow Value
   RUNG wire#powerrail
      Contact( #Always_On )
      Move(in := #"FT_Corrected Vol flow Val", out1 => #"Q_Corrected Vol flow Val")
   END_RUNG
   // the same network as SCL:
   IF #Always_On THEN #"Q_Corrected Vol flow Val" := #"FT_Corrected Vol flow Val"; END_IF;
END_REGION

REGION Network 8: FT_Corrected volume flow Status
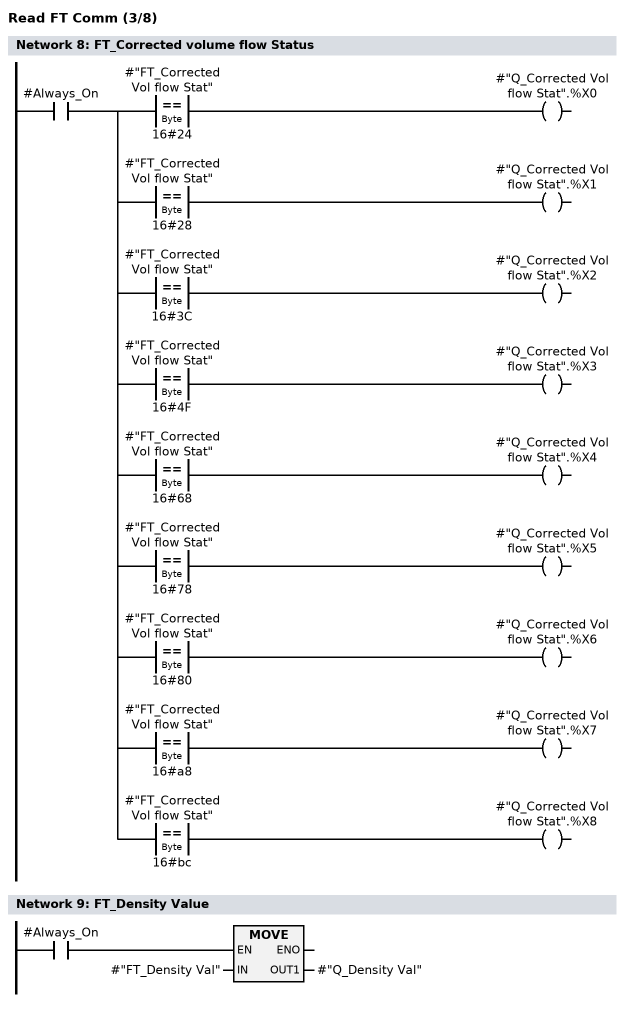
   RUNG wire#powerrail
      Contact( #Always_On )
      wire#w1
      { S7_Templates := "SrcType := Byte" } EQ_Contact(in1 := #"FT_Corrected Vol flow Stat", in2 := 16#24)
      Coil( #"Q_Corrected Vol flow Stat".%X0 )
   END_RUNG
   RUNG wire#w1
      { S7_Templates := "SrcType := Byte" } EQ_Contact(in1 := #"FT_Corrected Vol flow Stat", in2 := 16#28)
      Coil( #"Q_Corrected Vol flow Stat".%X1 )
   END_RUNG
   RUNG wire#w1
      { S7_Templates := "SrcType := Byte" } EQ_Contact(in1 := #"FT_Corrected Vol flow Stat", in2 := 16#3C)
      Coil( #"Q_Corrected Vol flow Stat".%X2 )
   END_RUNG
   RUNG wire#w1
      { S7_Templates := "SrcType := Byte" } EQ_Contact(in1 := #"FT_Corrected Vol flow Stat", in2 := 16#4F)
      Coil( #"Q_Corrected Vol flow Stat".%X3 )
   END_RUNG
   RUNG wire#w1
      { S7_Templates := "SrcType := Byte" } EQ_Contact(in1 := #"FT_Corrected Vol flow Stat", in2 := 16#68)
      Coil( #"Q_Corrected Vol flow Stat".%X4 )
   END_RUNG
   RUNG wire#w1
      { S7_Templates := "SrcType := Byte" } EQ_Contact(in1 := #"FT_Corrected Vol flow Stat", in2 := 16#78)
      Coil( #"Q_Corrected Vol flow Stat".%X5 )
   END_RUNG
   RUNG wire#w1
      { S7_Templates := "SrcType := Byte" } EQ_Contact(in1 := #"FT_Corrected Vol flow Stat", in2 := 16#80)
      Coil( #"Q_Corrected Vol flow Stat".%X6 )
   END_RUNG
   RUNG wire#w1
      { S7_Templates := "SrcType := Byte" } EQ_Contact(in1 := #"FT_Corrected Vol flow Stat", in2 := 16#a8)
      Coil( #"Q_Corrected Vol flow Stat".%X7 )
   END_RUNG
   RUNG wire#w1
      { S7_Templates := "SrcType := Byte" } EQ_Contact(in1 := #"FT_Corrected Vol flow Stat", in2 := 16#bc)
      Coil( #"Q_Corrected Vol flow Stat".%X8 )
   END_RUNG
   // the same network as SCL:
   #"Q_Corrected Vol flow Stat".%X0 := #Always_On AND (#"FT_Corrected Vol flow Stat" = 16#24);
   #"Q_Corrected Vol flow Stat".%X1 := #Always_On AND (#"FT_Corrected Vol flow Stat" = 16#28);
   #"Q_Corrected Vol flow Stat".%X2 := #Always_On AND (#"FT_Corrected Vol flow Stat" = 16#3C);
   #"Q_Corrected Vol flow Stat".%X3 := #Always_On AND (#"FT_Corrected Vol flow Stat" = 16#4F);
   #"Q_Corrected Vol flow Stat".%X4 := #Always_On AND (#"FT_Corrected Vol flow Stat" = 16#68);
   #"Q_Corrected Vol flow Stat".%X5 := #Always_On AND (#"FT_Corrected Vol flow Stat" = 16#78);
   #"Q_Corrected Vol flow Stat".%X6 := #Always_On AND (#"FT_Corrected Vol flow Stat" = 16#80);
   #"Q_Corrected Vol flow Stat".%X7 := #Always_On AND (#"FT_Corrected Vol flow Stat" = 16#a8);
   #"Q_Corrected Vol flow Stat".%X8 := #Always_On AND (#"FT_Corrected Vol flow Stat" = 16#bc);
END_REGION

REGION Network 9: FT_Density Value
   RUNG wire#powerrail
      Contact( #Always_On )
      Move(in := #"FT_Density Val", out1 => #"Q_Density Val")
   END_RUNG
   // the same network as SCL:
   IF #Always_On THEN #"Q_Density Val" := #"FT_Density Val"; END_IF;
END_REGION

REGION Network 10: FT_Density Status
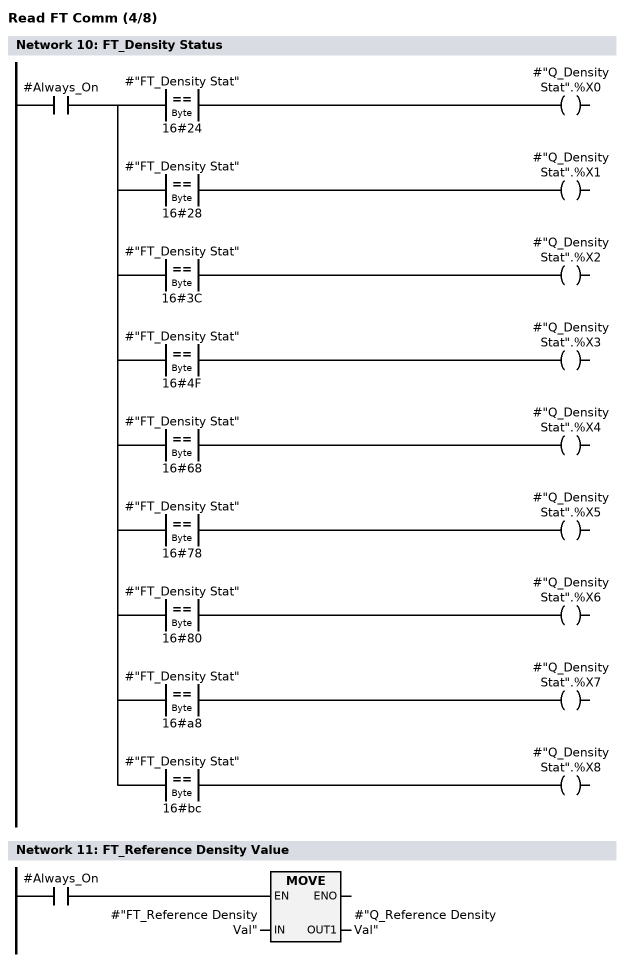
   RUNG wire#powerrail
      Contact( #Always_On )
      wire#w1
      { S7_Templates := "SrcType := Byte" } EQ_Contact(in1 := #"FT_Density Stat", in2 := 16#24)
      Coil( #"Q_Density Stat".%X0 )
   END_RUNG
   RUNG wire#w1
      { S7_Templates := "SrcType := Byte" } EQ_Contact(in1 := #"FT_Density Stat", in2 := 16#28)
      Coil( #"Q_Density Stat".%X1 )
   END_RUNG
   RUNG wire#w1
      { S7_Templates := "SrcType := Byte" } EQ_Contact(in1 := #"FT_Density Stat", in2 := 16#3C)
      Coil( #"Q_Density Stat".%X2 )
   END_RUNG
   RUNG wire#w1
      { S7_Templates := "SrcType := Byte" } EQ_Contact(in1 := #"FT_Density Stat", in2 := 16#4F)
      Coil( #"Q_Density Stat".%X3 )
   END_RUNG
   RUNG wire#w1
      { S7_Templates := "SrcType := Byte" } EQ_Contact(in1 := #"FT_Density Stat", in2 := 16#68)
      Coil( #"Q_Density Stat".%X4 )
   END_RUNG
   RUNG wire#w1
      { S7_Templates := "SrcType := Byte" } EQ_Contact(in1 := #"FT_Density Stat", in2 := 16#78)
      Coil( #"Q_Density Stat".%X5 )
   END_RUNG
   RUNG wire#w1
      { S7_Templates := "SrcType := Byte" } EQ_Contact(in1 := #"FT_Density Stat", in2 := 16#80)
      Coil( #"Q_Density Stat".%X6 )
   END_RUNG
   RUNG wire#w1
      { S7_Templates := "SrcType := Byte" } EQ_Contact(in1 := #"FT_Density Stat", in2 := 16#a8)
      Coil( #"Q_Density Stat".%X7 )
   END_RUNG
   RUNG wire#w1
      { S7_Templates := "SrcType := Byte" } EQ_Contact(in1 := #"FT_Density Stat", in2 := 16#bc)
      Coil( #"Q_Density Stat".%X8 )
   END_RUNG
   // the same network as SCL:
   #"Q_Density Stat".%X0 := #Always_On AND (#"FT_Density Stat" = 16#24);
   #"Q_Density Stat".%X1 := #Always_On AND (#"FT_Density Stat" = 16#28);
   #"Q_Density Stat".%X2 := #Always_On AND (#"FT_Density Stat" = 16#3C);
   #"Q_Density Stat".%X3 := #Always_On AND (#"FT_Density Stat" = 16#4F);
   #"Q_Density Stat".%X4 := #Always_On AND (#"FT_Density Stat" = 16#68);
   #"Q_Density Stat".%X5 := #Always_On AND (#"FT_Density Stat" = 16#78);
   #"Q_Density Stat".%X6 := #Always_On AND (#"FT_Density Stat" = 16#80);
   #"Q_Density Stat".%X7 := #Always_On AND (#"FT_Density Stat" = 16#a8);
   #"Q_Density Stat".%X8 := #Always_On AND (#"FT_Density Stat" = 16#bc);
END_REGION

REGION Network 11: FT_Reference Density Value
   RUNG wire#powerrail
      Contact( #Always_On )
      Move(in := #"FT_Reference Density Val", out1 => #"Q_Reference Density Val")
   END_RUNG
   // the same network as SCL:
   IF #Always_On THEN #"Q_Reference Density Val" := #"FT_Reference Density Val"; END_IF;
END_REGION

REGION Network 12: FT_Reference Density Status
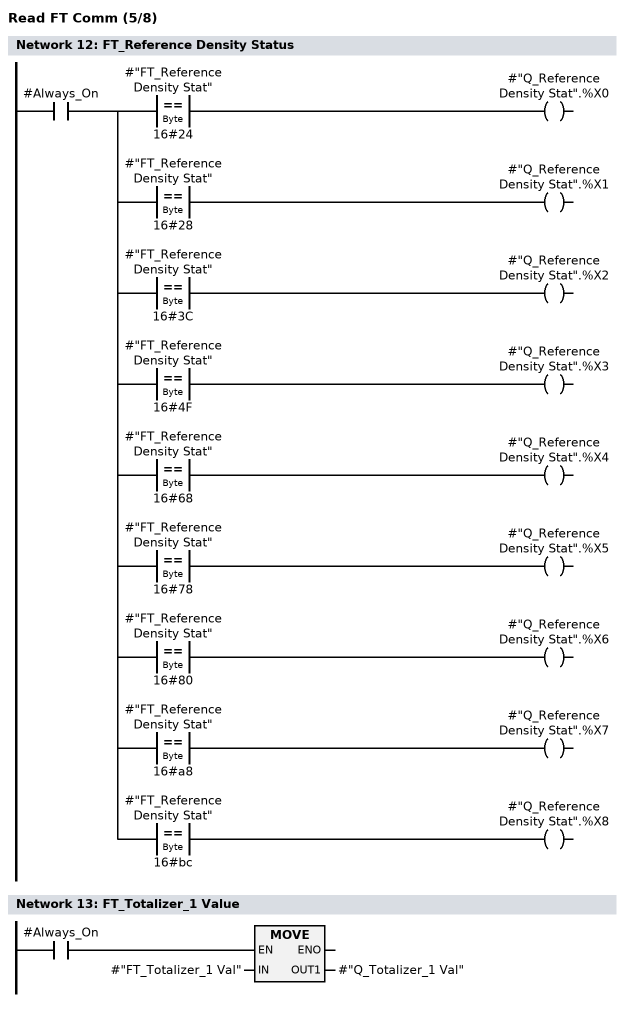
   RUNG wire#powerrail
      Contact( #Always_On )
      wire#w1
      { S7_Templates := "SrcType := Byte" } EQ_Contact(in1 := #"FT_Reference Density Stat", in2 := 16#24)
      Coil( #"Q_Reference Density Stat".%X0 )
   END_RUNG
   RUNG wire#w1
      { S7_Templates := "SrcType := Byte" } EQ_Contact(in1 := #"FT_Reference Density Stat", in2 := 16#28)
      Coil( #"Q_Reference Density Stat".%X1 )
   END_RUNG
   RUNG wire#w1
      { S7_Templates := "SrcType := Byte" } EQ_Contact(in1 := #"FT_Reference Density Stat", in2 := 16#3C)
      Coil( #"Q_Reference Density Stat".%X2 )
   END_RUNG
   RUNG wire#w1
      { S7_Templates := "SrcType := Byte" } EQ_Contact(in1 := #"FT_Reference Density Stat", in2 := 16#4F)
      Coil( #"Q_Reference Density Stat".%X3 )
   END_RUNG
   RUNG wire#w1
      { S7_Templates := "SrcType := Byte" } EQ_Contact(in1 := #"FT_Reference Density Stat", in2 := 16#68)
      Coil( #"Q_Reference Density Stat".%X4 )
   END_RUNG
   RUNG wire#w1
      { S7_Templates := "SrcType := Byte" } EQ_Contact(in1 := #"FT_Reference Density Stat", in2 := 16#78)
      Coil( #"Q_Reference Density Stat".%X5 )
   END_RUNG
   RUNG wire#w1
      { S7_Templates := "SrcType := Byte" } EQ_Contact(in1 := #"FT_Reference Density Stat", in2 := 16#80)
      Coil( #"Q_Reference Density Stat".%X6 )
   END_RUNG
   RUNG wire#w1
      { S7_Templates := "SrcType := Byte" } EQ_Contact(in1 := #"FT_Reference Density Stat", in2 := 16#a8)
      Coil( #"Q_Reference Density Stat".%X7 )
   END_RUNG
   RUNG wire#w1
      { S7_Templates := "SrcType := Byte" } EQ_Contact(in1 := #"FT_Reference Density Stat", in2 := 16#bc)
      Coil( #"Q_Reference Density Stat".%X8 )
   END_RUNG
   // the same network as SCL:
   #"Q_Reference Density Stat".%X0 := #Always_On AND (#"FT_Reference Density Stat" = 16#24);
   #"Q_Reference Density Stat".%X1 := #Always_On AND (#"FT_Reference Density Stat" = 16#28);
   #"Q_Reference Density Stat".%X2 := #Always_On AND (#"FT_Reference Density Stat" = 16#3C);
   #"Q_Reference Density Stat".%X3 := #Always_On AND (#"FT_Reference Density Stat" = 16#4F);
   #"Q_Reference Density Stat".%X4 := #Always_On AND (#"FT_Reference Density Stat" = 16#68);
   #"Q_Reference Density Stat".%X5 := #Always_On AND (#"FT_Reference Density Stat" = 16#78);
   #"Q_Reference Density Stat".%X6 := #Always_On AND (#"FT_Reference Density Stat" = 16#80);
   #"Q_Reference Density Stat".%X7 := #Always_On AND (#"FT_Reference Density Stat" = 16#a8);
   #"Q_Reference Density Stat".%X8 := #Always_On AND (#"FT_Reference Density Stat" = 16#bc);
END_REGION

REGION Network 13: FT_Totalizer_1 Value
   RUNG wire#powerrail
      Contact( #Always_On )
      Move(in := #"FT_Totalizer_1 Val", out1 => #"Q_Totalizer_1 Val")
   END_RUNG
   // the same network as SCL:
   IF #Always_On THEN #"Q_Totalizer_1 Val" := #"FT_Totalizer_1 Val"; END_IF;
END_REGION

REGION Network 14: FT_Totalizer_1 Status
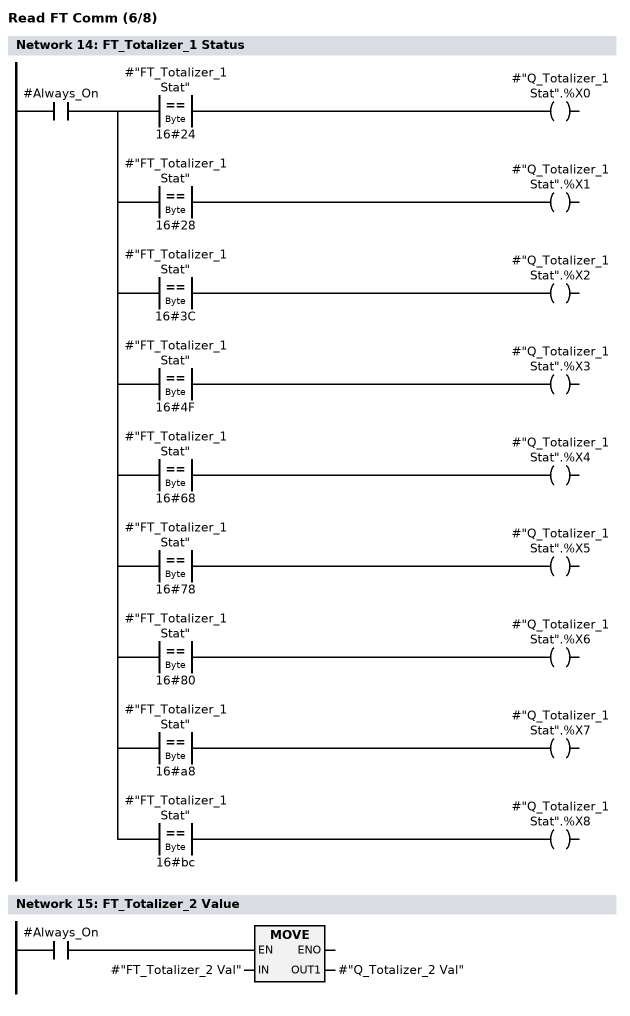
   RUNG wire#powerrail
      Contact( #Always_On )
      wire#w1
      { S7_Templates := "SrcType := Byte" } EQ_Contact(in1 := #"FT_Totalizer_1 Stat", in2 := 16#24)
      Coil( #"Q_Totalizer_1 Stat".%X0 )
   END_RUNG
   RUNG wire#w1
      { S7_Templates := "SrcType := Byte" } EQ_Contact(in1 := #"FT_Totalizer_1 Stat", in2 := 16#28)
      Coil( #"Q_Totalizer_1 Stat".%X1 )
   END_RUNG
   RUNG wire#w1
      { S7_Templates := "SrcType := Byte" } EQ_Contact(in1 := #"FT_Totalizer_1 Stat", in2 := 16#3C)
      Coil( #"Q_Totalizer_1 Stat".%X2 )
   END_RUNG
   RUNG wire#w1
      { S7_Templates := "SrcType := Byte" } EQ_Contact(in1 := #"FT_Totalizer_1 Stat", in2 := 16#4F)
      Coil( #"Q_Totalizer_1 Stat".%X3 )
   END_RUNG
   RUNG wire#w1
      { S7_Templates := "SrcType := Byte" } EQ_Contact(in1 := #"FT_Totalizer_1 Stat", in2 := 16#68)
      Coil( #"Q_Totalizer_1 Stat".%X4 )
   END_RUNG
   RUNG wire#w1
      { S7_Templates := "SrcType := Byte" } EQ_Contact(in1 := #"FT_Totalizer_1 Stat", in2 := 16#78)
      Coil( #"Q_Totalizer_1 Stat".%X5 )
   END_RUNG
   RUNG wire#w1
      { S7_Templates := "SrcType := Byte" } EQ_Contact(in1 := #"FT_Totalizer_1 Stat", in2 := 16#80)
      Coil( #"Q_Totalizer_1 Stat".%X6 )
   END_RUNG
   RUNG wire#w1
      { S7_Templates := "SrcType := Byte" } EQ_Contact(in1 := #"FT_Totalizer_1 Stat", in2 := 16#a8)
      Coil( #"Q_Totalizer_1 Stat".%X7 )
   END_RUNG
   RUNG wire#w1
      { S7_Templates := "SrcType := Byte" } EQ_Contact(in1 := #"FT_Totalizer_1 Stat", in2 := 16#bc)
      Coil( #"Q_Totalizer_1 Stat".%X8 )
   END_RUNG
   // the same network as SCL:
   #"Q_Totalizer_1 Stat".%X0 := #Always_On AND (#"FT_Totalizer_1 Stat" = 16#24);
   #"Q_Totalizer_1 Stat".%X1 := #Always_On AND (#"FT_Totalizer_1 Stat" = 16#28);
   #"Q_Totalizer_1 Stat".%X2 := #Always_On AND (#"FT_Totalizer_1 Stat" = 16#3C);
   #"Q_Totalizer_1 Stat".%X3 := #Always_On AND (#"FT_Totalizer_1 Stat" = 16#4F);
   #"Q_Totalizer_1 Stat".%X4 := #Always_On AND (#"FT_Totalizer_1 Stat" = 16#68);
   #"Q_Totalizer_1 Stat".%X5 := #Always_On AND (#"FT_Totalizer_1 Stat" = 16#78);
   #"Q_Totalizer_1 Stat".%X6 := #Always_On AND (#"FT_Totalizer_1 Stat" = 16#80);
   #"Q_Totalizer_1 Stat".%X7 := #Always_On AND (#"FT_Totalizer_1 Stat" = 16#a8);
   #"Q_Totalizer_1 Stat".%X8 := #Always_On AND (#"FT_Totalizer_1 Stat" = 16#bc);
END_REGION

REGION Network 15: FT_Totalizer_2 Value
   RUNG wire#powerrail
      Contact( #Always_On )
      Move(in := #"FT_Totalizer_2 Val", out1 => #"Q_Totalizer_2 Val")
   END_RUNG
   // the same network as SCL:
   IF #Always_On THEN #"Q_Totalizer_2 Val" := #"FT_Totalizer_2 Val"; END_IF;
END_REGION

REGION Network 16: FT_Totalizer_2 Status
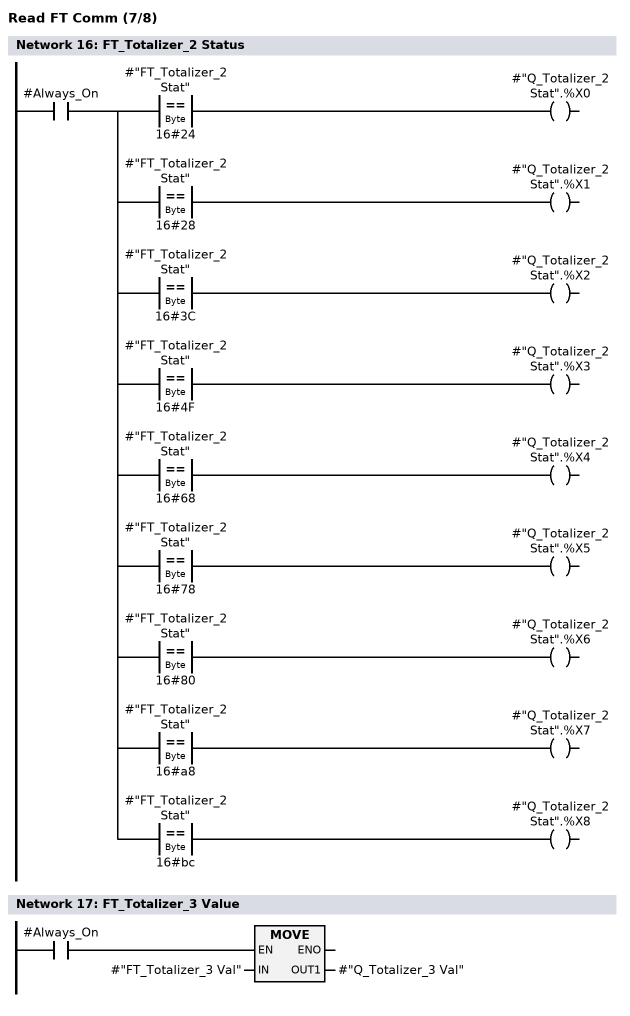
   RUNG wire#powerrail
      Contact( #Always_On )
      wire#w1
      { S7_Templates := "SrcType := Byte" } EQ_Contact(in1 := #"FT_Totalizer_2 Stat", in2 := 16#24)
      Coil( #"Q_Totalizer_2 Stat".%X0 )
   END_RUNG
   RUNG wire#w1
      { S7_Templates := "SrcType := Byte" } EQ_Contact(in1 := #"FT_Totalizer_2 Stat", in2 := 16#28)
      Coil( #"Q_Totalizer_2 Stat".%X1 )
   END_RUNG
   RUNG wire#w1
      { S7_Templates := "SrcType := Byte" } EQ_Contact(in1 := #"FT_Totalizer_2 Stat", in2 := 16#3C)
      Coil( #"Q_Totalizer_2 Stat".%X2 )
   END_RUNG
   RUNG wire#w1
      { S7_Templates := "SrcType := Byte" } EQ_Contact(in1 := #"FT_Totalizer_2 Stat", in2 := 16#4F)
      Coil( #"Q_Totalizer_2 Stat".%X3 )
   END_RUNG
   RUNG wire#w1
      { S7_Templates := "SrcType := Byte" } EQ_Contact(in1 := #"FT_Totalizer_2 Stat", in2 := 16#68)
      Coil( #"Q_Totalizer_2 Stat".%X4 )
   END_RUNG
   RUNG wire#w1
      { S7_Templates := "SrcType := Byte" } EQ_Contact(in1 := #"FT_Totalizer_2 Stat", in2 := 16#78)
      Coil( #"Q_Totalizer_2 Stat".%X5 )
   END_RUNG
   RUNG wire#w1
      { S7_Templates := "SrcType := Byte" } EQ_Contact(in1 := #"FT_Totalizer_2 Stat", in2 := 16#80)
      Coil( #"Q_Totalizer_2 Stat".%X6 )
   END_RUNG
   RUNG wire#w1
      { S7_Templates := "SrcType := Byte" } EQ_Contact(in1 := #"FT_Totalizer_2 Stat", in2 := 16#a8)
      Coil( #"Q_Totalizer_2 Stat".%X7 )
   END_RUNG
   RUNG wire#w1
      { S7_Templates := "SrcType := Byte" } EQ_Contact(in1 := #"FT_Totalizer_2 Stat", in2 := 16#bc)
      Coil( #"Q_Totalizer_2 Stat".%X8 )
   END_RUNG
   // the same network as SCL:
   #"Q_Totalizer_2 Stat".%X0 := #Always_On AND (#"FT_Totalizer_2 Stat" = 16#24);
   #"Q_Totalizer_2 Stat".%X1 := #Always_On AND (#"FT_Totalizer_2 Stat" = 16#28);
   #"Q_Totalizer_2 Stat".%X2 := #Always_On AND (#"FT_Totalizer_2 Stat" = 16#3C);
   #"Q_Totalizer_2 Stat".%X3 := #Always_On AND (#"FT_Totalizer_2 Stat" = 16#4F);
   #"Q_Totalizer_2 Stat".%X4 := #Always_On AND (#"FT_Totalizer_2 Stat" = 16#68);
   #"Q_Totalizer_2 Stat".%X5 := #Always_On AND (#"FT_Totalizer_2 Stat" = 16#78);
   #"Q_Totalizer_2 Stat".%X6 := #Always_On AND (#"FT_Totalizer_2 Stat" = 16#80);
   #"Q_Totalizer_2 Stat".%X7 := #Always_On AND (#"FT_Totalizer_2 Stat" = 16#a8);
   #"Q_Totalizer_2 Stat".%X8 := #Always_On AND (#"FT_Totalizer_2 Stat" = 16#bc);
END_REGION

REGION Network 17: FT_Totalizer_3 Value
   RUNG wire#powerrail
      Contact( #Always_On )
      Move(in := #"FT_Totalizer_3 Val", out1 => #"Q_Totalizer_3 Val")
   END_RUNG
   // the same network as SCL:
   IF #Always_On THEN #"Q_Totalizer_3 Val" := #"FT_Totalizer_3 Val"; END_IF;
END_REGION

REGION Network 18: FT_Totalizer_3 Status
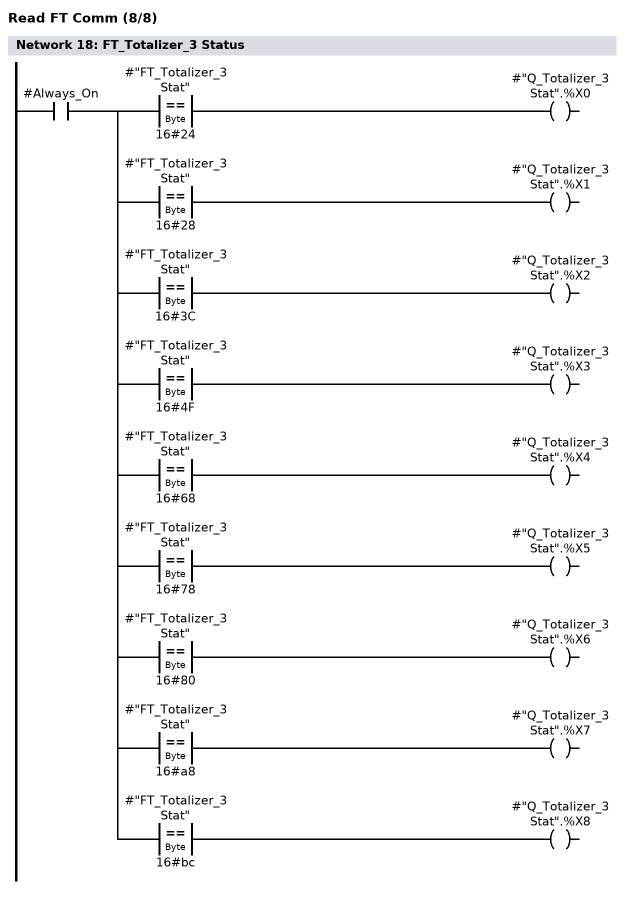
   RUNG wire#powerrail
      Contact( #Always_On )
      wire#w1
      { S7_Templates := "SrcType := Byte" } EQ_Contact(in1 := #"FT_Totalizer_3 Stat", in2 := 16#24)
      Coil( #"Q_Totalizer_3 Stat".%X0 )
   END_RUNG
   RUNG wire#w1
      { S7_Templates := "SrcType := Byte" } EQ_Contact(in1 := #"FT_Totalizer_3 Stat", in2 := 16#28)
      Coil( #"Q_Totalizer_3 Stat".%X1 )
   END_RUNG
   RUNG wire#w1
      { S7_Templates := "SrcType := Byte" } EQ_Contact(in1 := #"FT_Totalizer_3 Stat", in2 := 16#3C)
      Coil( #"Q_Totalizer_3 Stat".%X2 )
   END_RUNG
   RUNG wire#w1
      { S7_Templates := "SrcType := Byte" } EQ_Contact(in1 := #"FT_Totalizer_3 Stat", in2 := 16#4F)
      Coil( #"Q_Totalizer_3 Stat".%X3 )
   END_RUNG
   RUNG wire#w1
      { S7_Templates := "SrcType := Byte" } EQ_Contact(in1 := #"FT_Totalizer_3 Stat", in2 := 16#68)
      Coil( #"Q_Totalizer_3 Stat".%X4 )
   END_RUNG
   RUNG wire#w1
      { S7_Templates := "SrcType := Byte" } EQ_Contact(in1 := #"FT_Totalizer_3 Stat", in2 := 16#78)
      Coil( #"Q_Totalizer_3 Stat".%X5 )
   END_RUNG
   RUNG wire#w1
      { S7_Templates := "SrcType := Byte" } EQ_Contact(in1 := #"FT_Totalizer_3 Stat", in2 := 16#80)
      Coil( #"Q_Totalizer_3 Stat".%X6 )
   END_RUNG
   RUNG wire#w1
      { S7_Templates := "SrcType := Byte" } EQ_Contact(in1 := #"FT_Totalizer_3 Stat", in2 := 16#a8)
      Coil( #"Q_Totalizer_3 Stat".%X7 )
   END_RUNG
   RUNG wire#w1
      { S7_Templates := "SrcType := Byte" } EQ_Contact(in1 := #"FT_Totalizer_3 Stat", in2 := 16#bc)
      Coil( #"Q_Totalizer_3 Stat".%X8 )
   END_RUNG
   // the same network as SCL:
   #"Q_Totalizer_3 Stat".%X0 := #Always_On AND (#"FT_Totalizer_3 Stat" = 16#24);
   #"Q_Totalizer_3 Stat".%X1 := #Always_On AND (#"FT_Totalizer_3 Stat" = 16#28);
   #"Q_Totalizer_3 Stat".%X2 := #Always_On AND (#"FT_Totalizer_3 Stat" = 16#3C);
   #"Q_Totalizer_3 Stat".%X3 := #Always_On AND (#"FT_Totalizer_3 Stat" = 16#4F);
   #"Q_Totalizer_3 Stat".%X4 := #Always_On AND (#"FT_Totalizer_3 Stat" = 16#68);
   #"Q_Totalizer_3 Stat".%X5 := #Always_On AND (#"FT_Totalizer_3 Stat" = 16#78);
   #"Q_Totalizer_3 Stat".%X6 := #Always_On AND (#"FT_Totalizer_3 Stat" = 16#80);
   #"Q_Totalizer_3 Stat".%X7 := #Always_On AND (#"FT_Totalizer_3 Stat" = 16#a8);
   #"Q_Totalizer_3 Stat".%X8 := #Always_On AND (#"FT_Totalizer_3 Stat" = 16#bc);
END_REGION
END_FUNCTION_BLOCK

FUNCTION_BLOCK "IO Digital Preparation"   // FB8, LAD
{ S7_Optimized_Access := 'FALSE' }
VERSION : 0.1
// stored: AutoNumber true, IsIECCheckEnabled false, SetENOAutomatically false, UDAEnableTagReadback false
   VAR_INPUT
      init : Bool;
      Reset : Bool;
   END_VAR
   VAR
      "FS-01.01" { S7_SetPoint := 'True'} : "Digital";   // FLOW SWITCH LINE HOT WATER PHE-01.01
      "DRP-P02.01" { S7_SetPoint := 'True'} : "Digital";   // DRY RUN PROTECTION MONO PUMP P-02.01
      "DRP-P02.02" { S7_SetPoint := 'True'} : "Digital";   // DRY RUN PROTECTION MONO PUMP P-02.03
      "DRP-P03.01" { S7_SetPoint := 'True'} : "Digital";   // DRY RUN PROTECTION MONO PUMP P-03.01
      "DRP-P03.02" { S7_SetPoint := 'True'} : "Digital";   // DRY RUN PROTECTION MONO PUMP P-03.03
      "DRP-P04.01" { S7_SetPoint := 'True'} : "Digital";   // DRY RUN PROTECTION MONO PUMP P-04.01
      "DRP-P05.01" { S7_SetPoint := 'True'} : "Digital";   // DRY RUN PROTECTION MONO PUMP P-05.01
      "DRP-P05.02" { S7_SetPoint := 'True'} : "Digital";   // DRY RUN PROTECTION MONO PUMP P-05.03
      "DRP-P06.01" { S7_SetPoint := 'True'} : "Digital";   // DRY RUN PROTECTION MONO PUMP P-06.01
      "DRP-P07.01" { S7_SetPoint := 'True'} : "Digital";   // DRY RUN PROTECTION MONO PUMP P-07.01
      "DRP-P08.01" { S7_SetPoint := 'True'} : "Digital";   // DRY RUN PROTECTION MONO PUMP P-08.01
      "DRP-P09.01" { S7_SetPoint := 'True'} : "Digital";   // DRY RUN PROTECTION MONO PUMP P-09.01
      "DRP-P09.02" { S7_SetPoint := 'True'} : "Digital";   // DRY RUN PROTECTION MONO PUMP P-09.03
      "LL-51.01" { S7_SetPoint := 'True'} : "Digital";
      "ML-51.01" { S7_SetPoint := 'True'} : "Digital";
      "HL-51.01" { S7_SetPoint := 'True'} : "Digital";
   END_VAR
BEGIN

REGION Network 1: FS-01.01
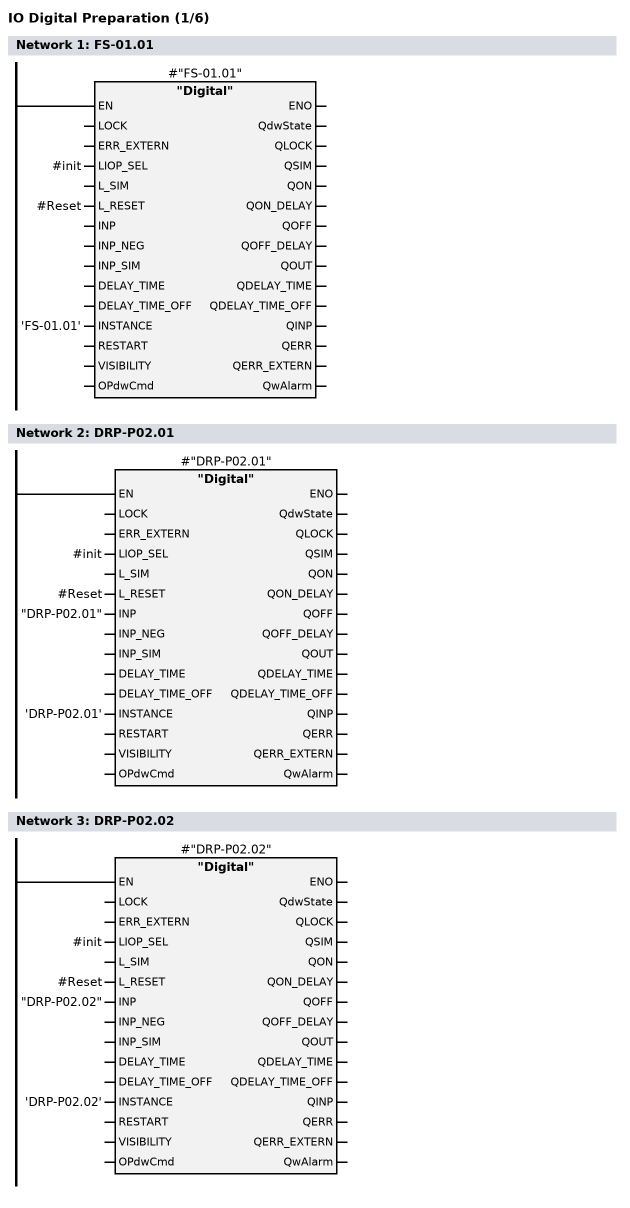
   RUNG wire#powerrail
      #"FS-01.01"(LOCK :=, ERR_EXTERN :=, LIOP_SEL := #init, L_SIM :=, L_RESET := #Reset, INP :=, INP_NEG :=, INP_SIM :=, DELAY_TIME :=, DELAY_TIME_OFF :=, INSTANCE := 'FS-01.01', RESTART :=, VISIBILITY :=, OPdwCmd :=, QdwState =>, QLOCK =>, QSIM =>, QON =>, QON_DELAY =>, QOFF =>, QOFF_DELAY =>, QOUT =>, QDELAY_TIME =>, QDELAY_TIME_OFF =>, QINP =>, QERR =>, QERR_EXTERN =>, QwAlarm =>)
   END_RUNG
   // the same network as SCL:
   #"FS-01.01"(LIOP_SEL := #init, L_RESET := #Reset, INSTANCE := 'FS-01.01');   // "Digital"
END_REGION

REGION Network 2: DRP-P02.01
   RUNG wire#powerrail
      #"DRP-P02.01"(LOCK :=, ERR_EXTERN :=, LIOP_SEL := #init, L_SIM :=, L_RESET := #Reset, INP := "DRP-P02.01", INP_NEG :=, INP_SIM :=, DELAY_TIME :=, DELAY_TIME_OFF :=, INSTANCE := 'DRP-P02.01', RESTART :=, VISIBILITY :=, OPdwCmd :=, QdwState =>, QLOCK =>, QSIM =>, QON =>, QON_DELAY =>, QOFF =>, QOFF_DELAY =>, QOUT =>, QDELAY_TIME =>, QDELAY_TIME_OFF =>, QINP =>, QERR =>, QERR_EXTERN =>, QwAlarm =>)
   END_RUNG
   // the same network as SCL:
   #"DRP-P02.01"(LIOP_SEL := #init, L_RESET := #Reset, INP := "DRP-P02.01", INSTANCE := 'DRP-P02.01');   // "Digital"
END_REGION

REGION Network 3: DRP-P02.02
   RUNG wire#powerrail
      #"DRP-P02.02"(LOCK :=, ERR_EXTERN :=, LIOP_SEL := #init, L_SIM :=, L_RESET := #Reset, INP := "DRP-P02.02", INP_NEG :=, INP_SIM :=, DELAY_TIME :=, DELAY_TIME_OFF :=, INSTANCE := 'DRP-P02.02', RESTART :=, VISIBILITY :=, OPdwCmd :=, QdwState =>, QLOCK =>, QSIM =>, QON =>, QON_DELAY =>, QOFF =>, QOFF_DELAY =>, QOUT =>, QDELAY_TIME =>, QDELAY_TIME_OFF =>, QINP =>, QERR =>, QERR_EXTERN =>, QwAlarm =>)
   END_RUNG
   // the same network as SCL:
   #"DRP-P02.02"(LIOP_SEL := #init, L_RESET := #Reset, INP := "DRP-P02.02", INSTANCE := 'DRP-P02.02');   // "Digital"
END_REGION

REGION Network 4: DRP-P03.01
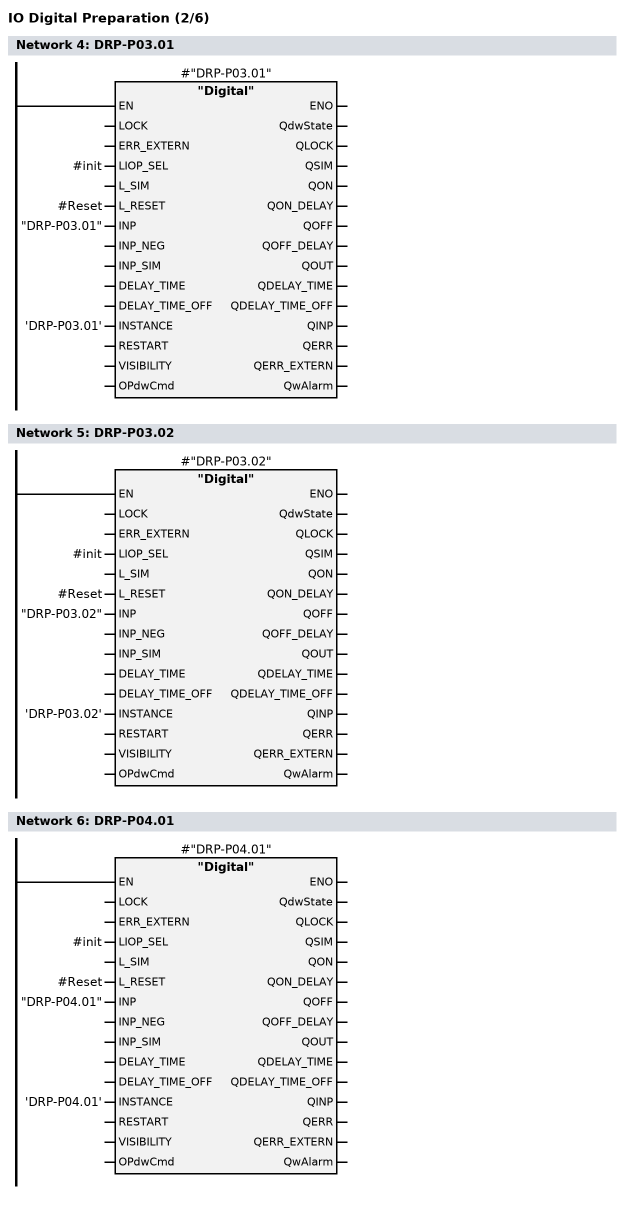
   RUNG wire#powerrail
      #"DRP-P03.01"(LOCK :=, ERR_EXTERN :=, LIOP_SEL := #init, L_SIM :=, L_RESET := #Reset, INP := "DRP-P03.01", INP_NEG :=, INP_SIM :=, DELAY_TIME :=, DELAY_TIME_OFF :=, INSTANCE := 'DRP-P03.01', RESTART :=, VISIBILITY :=, OPdwCmd :=, QdwState =>, QLOCK =>, QSIM =>, QON =>, QON_DELAY =>, QOFF =>, QOFF_DELAY =>, QOUT =>, QDELAY_TIME =>, QDELAY_TIME_OFF =>, QINP =>, QERR =>, QERR_EXTERN =>, QwAlarm =>)
   END_RUNG
   // the same network as SCL:
   #"DRP-P03.01"(LIOP_SEL := #init, L_RESET := #Reset, INP := "DRP-P03.01", INSTANCE := 'DRP-P03.01');   // "Digital"
END_REGION

REGION Network 5: DRP-P03.02
   RUNG wire#powerrail
      #"DRP-P03.02"(LOCK :=, ERR_EXTERN :=, LIOP_SEL := #init, L_SIM :=, L_RESET := #Reset, INP := "DRP-P03.02", INP_NEG :=, INP_SIM :=, DELAY_TIME :=, DELAY_TIME_OFF :=, INSTANCE := 'DRP-P03.02', RESTART :=, VISIBILITY :=, OPdwCmd :=, QdwState =>, QLOCK =>, QSIM =>, QON =>, QON_DELAY =>, QOFF =>, QOFF_DELAY =>, QOUT =>, QDELAY_TIME =>, QDELAY_TIME_OFF =>, QINP =>, QERR =>, QERR_EXTERN =>, QwAlarm =>)
   END_RUNG
   // the same network as SCL:
   #"DRP-P03.02"(LIOP_SEL := #init, L_RESET := #Reset, INP := "DRP-P03.02", INSTANCE := 'DRP-P03.02');   // "Digital"
END_REGION

REGION Network 6: DRP-P04.01
   RUNG wire#powerrail
      #"DRP-P04.01"(LOCK :=, ERR_EXTERN :=, LIOP_SEL := #init, L_SIM :=, L_RESET := #Reset, INP := "DRP-P04.01", INP_NEG :=, INP_SIM :=, DELAY_TIME :=, DELAY_TIME_OFF :=, INSTANCE := 'DRP-P04.01', RESTART :=, VISIBILITY :=, OPdwCmd :=, QdwState =>, QLOCK =>, QSIM =>, QON =>, QON_DELAY =>, QOFF =>, QOFF_DELAY =>, QOUT =>, QDELAY_TIME =>, QDELAY_TIME_OFF =>, QINP =>, QERR =>, QERR_EXTERN =>, QwAlarm =>)
   END_RUNG
   // the same network as SCL:
   #"DRP-P04.01"(LIOP_SEL := #init, L_RESET := #Reset, INP := "DRP-P04.01", INSTANCE := 'DRP-P04.01');   // "Digital"
END_REGION

REGION Network 7: DRP-P05.01
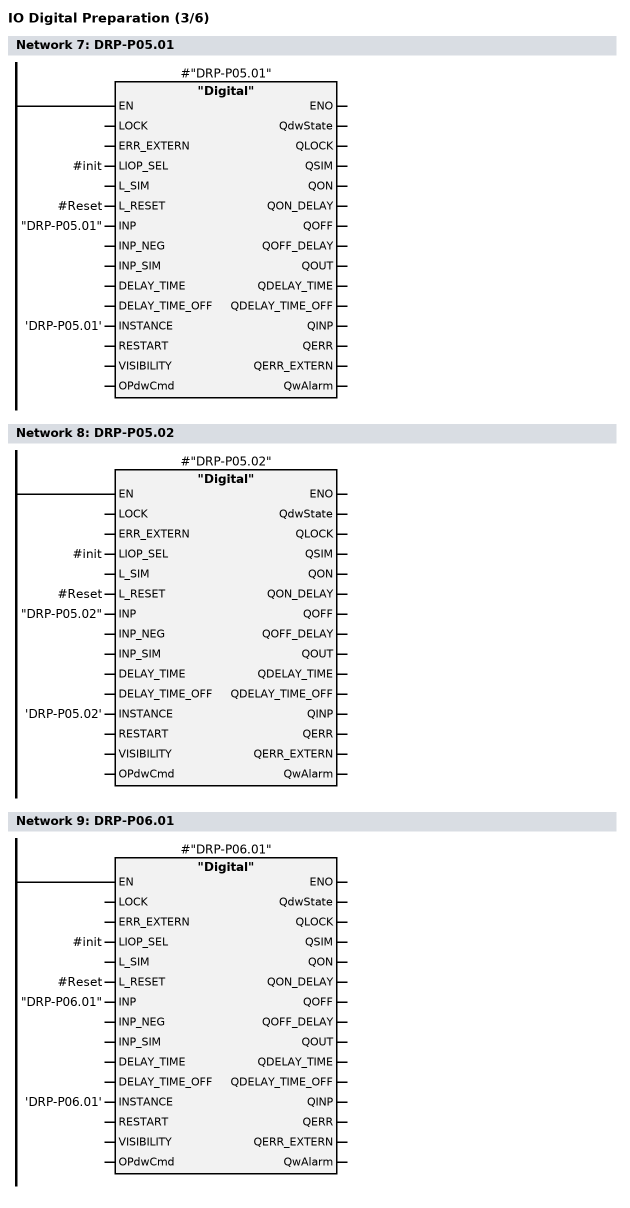
   RUNG wire#powerrail
      #"DRP-P05.01"(LOCK :=, ERR_EXTERN :=, LIOP_SEL := #init, L_SIM :=, L_RESET := #Reset, INP := "DRP-P05.01", INP_NEG :=, INP_SIM :=, DELAY_TIME :=, DELAY_TIME_OFF :=, INSTANCE := 'DRP-P05.01', RESTART :=, VISIBILITY :=, OPdwCmd :=, QdwState =>, QLOCK =>, QSIM =>, QON =>, QON_DELAY =>, QOFF =>, QOFF_DELAY =>, QOUT =>, QDELAY_TIME =>, QDELAY_TIME_OFF =>, QINP =>, QERR =>, QERR_EXTERN =>, QwAlarm =>)
   END_RUNG
   // the same network as SCL:
   #"DRP-P05.01"(LIOP_SEL := #init, L_RESET := #Reset, INP := "DRP-P05.01", INSTANCE := 'DRP-P05.01');   // "Digital"
END_REGION

REGION Network 8: DRP-P05.02
   RUNG wire#powerrail
      #"DRP-P05.02"(LOCK :=, ERR_EXTERN :=, LIOP_SEL := #init, L_SIM :=, L_RESET := #Reset, INP := "DRP-P05.02", INP_NEG :=, INP_SIM :=, DELAY_TIME :=, DELAY_TIME_OFF :=, INSTANCE := 'DRP-P05.02', RESTART :=, VISIBILITY :=, OPdwCmd :=, QdwState =>, QLOCK =>, QSIM =>, QON =>, QON_DELAY =>, QOFF =>, QOFF_DELAY =>, QOUT =>, QDELAY_TIME =>, QDELAY_TIME_OFF =>, QINP =>, QERR =>, QERR_EXTERN =>, QwAlarm =>)
   END_RUNG
   // the same network as SCL:
   #"DRP-P05.02"(LIOP_SEL := #init, L_RESET := #Reset, INP := "DRP-P05.02", INSTANCE := 'DRP-P05.02');   // "Digital"
END_REGION

REGION Network 9: DRP-P06.01
   RUNG wire#powerrail
      #"DRP-P06.01"(LOCK :=, ERR_EXTERN :=, LIOP_SEL := #init, L_SIM :=, L_RESET := #Reset, INP := "DRP-P06.01", INP_NEG :=, INP_SIM :=, DELAY_TIME :=, DELAY_TIME_OFF :=, INSTANCE := 'DRP-P06.01', RESTART :=, VISIBILITY :=, OPdwCmd :=, QdwState =>, QLOCK =>, QSIM =>, QON =>, QON_DELAY =>, QOFF =>, QOFF_DELAY =>, QOUT =>, QDELAY_TIME =>, QDELAY_TIME_OFF =>, QINP =>, QERR =>, QERR_EXTERN =>, QwAlarm =>)
   END_RUNG
   // the same network as SCL:
   #"DRP-P06.01"(LIOP_SEL := #init, L_RESET := #Reset, INP := "DRP-P06.01", INSTANCE := 'DRP-P06.01');   // "Digital"
END_REGION

REGION Network 10: DRP-P07.01
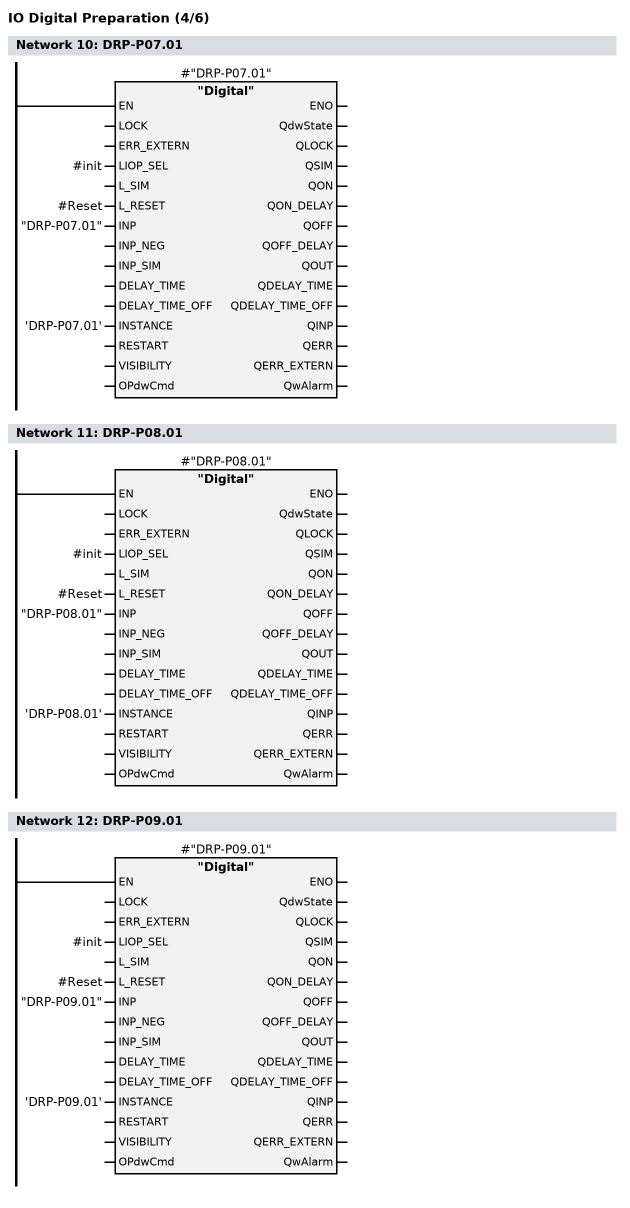
   RUNG wire#powerrail
      #"DRP-P07.01"(LOCK :=, ERR_EXTERN :=, LIOP_SEL := #init, L_SIM :=, L_RESET := #Reset, INP := "DRP-P07.01", INP_NEG :=, INP_SIM :=, DELAY_TIME :=, DELAY_TIME_OFF :=, INSTANCE := 'DRP-P07.01', RESTART :=, VISIBILITY :=, OPdwCmd :=, QdwState =>, QLOCK =>, QSIM =>, QON =>, QON_DELAY =>, QOFF =>, QOFF_DELAY =>, QOUT =>, QDELAY_TIME =>, QDELAY_TIME_OFF =>, QINP =>, QERR =>, QERR_EXTERN =>, QwAlarm =>)
   END_RUNG
   // the same network as SCL:
   #"DRP-P07.01"(LIOP_SEL := #init, L_RESET := #Reset, INP := "DRP-P07.01", INSTANCE := 'DRP-P07.01');   // "Digital"
END_REGION

REGION Network 11: DRP-P08.01
   RUNG wire#powerrail
      #"DRP-P08.01"(LOCK :=, ERR_EXTERN :=, LIOP_SEL := #init, L_SIM :=, L_RESET := #Reset, INP := "DRP-P08.01", INP_NEG :=, INP_SIM :=, DELAY_TIME :=, DELAY_TIME_OFF :=, INSTANCE := 'DRP-P08.01', RESTART :=, VISIBILITY :=, OPdwCmd :=, QdwState =>, QLOCK =>, QSIM =>, QON =>, QON_DELAY =>, QOFF =>, QOFF_DELAY =>, QOUT =>, QDELAY_TIME =>, QDELAY_TIME_OFF =>, QINP =>, QERR =>, QERR_EXTERN =>, QwAlarm =>)
   END_RUNG
   // the same network as SCL:
   #"DRP-P08.01"(LIOP_SEL := #init, L_RESET := #Reset, INP := "DRP-P08.01", INSTANCE := 'DRP-P08.01');   // "Digital"
END_REGION

REGION Network 12: DRP-P09.01
   RUNG wire#powerrail
      #"DRP-P09.01"(LOCK :=, ERR_EXTERN :=, LIOP_SEL := #init, L_SIM :=, L_RESET := #Reset, INP := "DRP-P09.01", INP_NEG :=, INP_SIM :=, DELAY_TIME :=, DELAY_TIME_OFF :=, INSTANCE := 'DRP-P09.01', RESTART :=, VISIBILITY :=, OPdwCmd :=, QdwState =>, QLOCK =>, QSIM =>, QON =>, QON_DELAY =>, QOFF =>, QOFF_DELAY =>, QOUT =>, QDELAY_TIME =>, QDELAY_TIME_OFF =>, QINP =>, QERR =>, QERR_EXTERN =>, QwAlarm =>)
   END_RUNG
   // the same network as SCL:
   #"DRP-P09.01"(LIOP_SEL := #init, L_RESET := #Reset, INP := "DRP-P09.01", INSTANCE := 'DRP-P09.01');   // "Digital"
END_REGION

REGION Network 13: DRP-P09.02
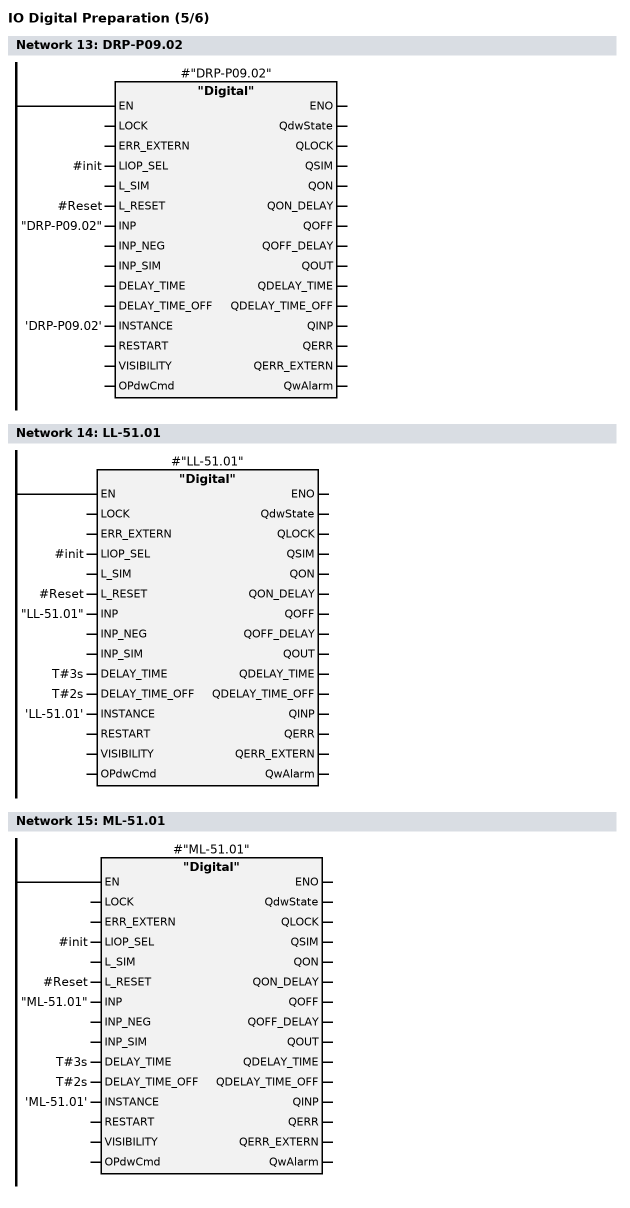
   RUNG wire#powerrail
      #"DRP-P09.02"(LOCK :=, ERR_EXTERN :=, LIOP_SEL := #init, L_SIM :=, L_RESET := #Reset, INP := "DRP-P09.02", INP_NEG :=, INP_SIM :=, DELAY_TIME :=, DELAY_TIME_OFF :=, INSTANCE := 'DRP-P09.02', RESTART :=, VISIBILITY :=, OPdwCmd :=, QdwState =>, QLOCK =>, QSIM =>, QON =>, QON_DELAY =>, QOFF =>, QOFF_DELAY =>, QOUT =>, QDELAY_TIME =>, QDELAY_TIME_OFF =>, QINP =>, QERR =>, QERR_EXTERN =>, QwAlarm =>)
   END_RUNG
   // the same network as SCL:
   #"DRP-P09.02"(LIOP_SEL := #init, L_RESET := #Reset, INP := "DRP-P09.02", INSTANCE := 'DRP-P09.02');   // "Digital"
END_REGION

REGION Network 14: LL-51.01
   RUNG wire#powerrail
      #"LL-51.01"(LOCK :=, ERR_EXTERN :=, LIOP_SEL := #init, L_SIM :=, L_RESET := #Reset, INP := "LL-51.01", INP_NEG :=, INP_SIM :=, DELAY_TIME := T#3s, DELAY_TIME_OFF := T#2s, INSTANCE := 'LL-51.01', RESTART :=, VISIBILITY :=, OPdwCmd :=, QdwState =>, QLOCK =>, QSIM =>, QON =>, QON_DELAY =>, QOFF =>, QOFF_DELAY =>, QOUT =>, QDELAY_TIME =>, QDELAY_TIME_OFF =>, QINP =>, QERR =>, QERR_EXTERN =>, QwAlarm =>)
   END_RUNG
   // the same network as SCL:
   #"LL-51.01"(LIOP_SEL := #init,   // "Digital"
               L_RESET := #Reset,
               INP := "LL-51.01",
               DELAY_TIME := T#3s,
               DELAY_TIME_OFF := T#2s,
               INSTANCE := 'LL-51.01');
END_REGION

REGION Network 15: ML-51.01
   RUNG wire#powerrail
      #"ML-51.01"(LOCK :=, ERR_EXTERN :=, LIOP_SEL := #init, L_SIM :=, L_RESET := #Reset, INP := "ML-51.01", INP_NEG :=, INP_SIM :=, DELAY_TIME := T#3s, DELAY_TIME_OFF := T#2s, INSTANCE := 'ML-51.01', RESTART :=, VISIBILITY :=, OPdwCmd :=, QdwState =>, QLOCK =>, QSIM =>, QON =>, QON_DELAY =>, QOFF =>, QOFF_DELAY =>, QOUT =>, QDELAY_TIME =>, QDELAY_TIME_OFF =>, QINP =>, QERR =>, QERR_EXTERN =>, QwAlarm =>)
   END_RUNG
   // the same network as SCL:
   #"ML-51.01"(LIOP_SEL := #init,   // "Digital"
               L_RESET := #Reset,
               INP := "ML-51.01",
               DELAY_TIME := T#3s,
               DELAY_TIME_OFF := T#2s,
               INSTANCE := 'ML-51.01');
END_REGION

REGION Network 16: HL-51.01
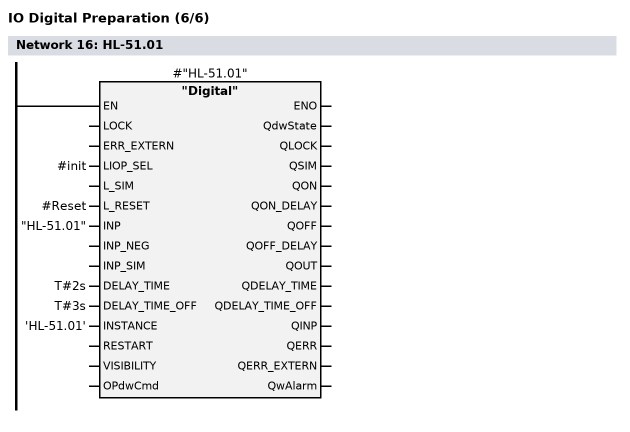
   RUNG wire#powerrail
      #"HL-51.01"(LOCK :=, ERR_EXTERN :=, LIOP_SEL := #init, L_SIM :=, L_RESET := #Reset, INP := "HL-51.01", INP_NEG :=, INP_SIM :=, DELAY_TIME := T#2s, DELAY_TIME_OFF := T#3s, INSTANCE := 'HL-51.01', RESTART :=, VISIBILITY :=, OPdwCmd :=, QdwState =>, QLOCK =>, QSIM =>, QON =>, QON_DELAY =>, QOFF =>, QOFF_DELAY =>, QOUT =>, QDELAY_TIME =>, QDELAY_TIME_OFF =>, QINP =>, QERR =>, QERR_EXTERN =>, QwAlarm =>)
   END_RUNG
   // the same network as SCL:
   #"HL-51.01"(LIOP_SEL := #init,   // "Digital"
               L_RESET := #Reset,
               INP := "HL-51.01",
               DELAY_TIME := T#2s,
               DELAY_TIME_OFF := T#3s,
               INSTANCE := 'HL-51.01');
END_REGION
END_FUNCTION_BLOCK

FUNCTION_BLOCK "Digital"
TITLE =  Digital
{ S7_Optimized_Access := 'FALSE' }
AUTHOR : RM
FAMILY : MON
VERSION : 0.1
//Interface for a binary value  
   VAR_INPUT 
      LOCK : Bool;   // 1 = Inerlock active
      ERR_EXTERN : Bool;   // 1 = External error arised
      LIOP_SEL : Bool;   // 0 = Operator; 1 = Linking
      L_SIM : Bool;   // 0 = Normal; 1 = Simulation
      L_RESET : Bool;   // 1 = Reset error peripherie
      INP : Bool;   // 1 = Digital input signal is ON
      INP_NEG : Bool;   // 1 = Negation input signal is ACTIVE
      INP_SIM : Bool;   // 1 = Digital simulation signal is ON
      DELAY_TIME : Time := T#5S;   // Delay time of setting bit
      DELAY_TIME_OFF : Time := T#5S;   // Delay time of resetting bit
      INSTANCE : String[254] := 'Digital_001';   // Filter attribute for message view, also used for labelling
      RESTART : Bool;   // 1 = Initialize FB at startup (first cycle fo PLC)
   END_VAR

   VAR_OUTPUT 
      QdwState : DWord;   // Status HMI
      QLOCK : Bool;   // 1 = Interlock is active
      QSIM : Bool;   // 0 = Normal; 1 = Simulation
      QON : Bool;   // 1 = On
      QON_DELAY : Bool;   // 1 = On with delay
      QOFF : Bool;   // 1 = Off
      QOFF_DELAY : Bool;   // 1 = Off with delay
      QOUT : Bool;   // 1 = On or 1 = Off with delay, DI Out with Time Delay
      QDELAY_TIME : Time;   // Delay time for switching ON
      QDELAY_TIME_OFF : Time;   // Delay time for switching OFF
      QINP : Bool;   // 1 = Input signal including negation information
      QERR : Bool;   // 1 = Common error
      QERR_EXTERN : Bool;   // 1 = External error
      QwAlarm : Word;   // Bit alarm producere
   END_VAR

   VAR_IN_OUT 
      VISIBILITY : Byte;   // Bit 0: Tab1 of window; Bit 1: Tab2 of window; ... ; Bit 7: Minimize
      OPdwCmd : DWord;   // Control word from HMI
   END_VAR

   VAR 
      OP_RESET : Bool;   // Reset error
      OP_VISIBILITY : Byte;   // Operator: Bit 0: Tab1 of window; Bit 1: Tab2 of window; ... ; Bit 7: Minimize
      VISIBILITY_OLD : Byte;   // Save last status of VISIBILITY
      DELAY_ON : Bool;   // Delay for switching ON required
      DELAY_OFF : Bool;   // Delay for switching OFF required
      SE_L_RESET_LINK : Bool;   // Signal edge for the reset input from linking
      SE_L_RESET_LINK_COND : Bool;   // Condition of signal edge
      SE_L_RESET_OP : Bool;   // Signal edge for the reset input from operator
      T_ON {InstructionName := 'TON_TIME'; LibVersion := '1.0'} : TON_TIME;
      T_OFF {InstructionName := 'TON_TIME'; LibVersion := '1.0'} : TON_TIME;   // Timer instance for turning off
      OLD_SIG_COND : Bool;   // Condition of the old signal
      SINP_SIM : Bool;   // Signal from operator in simulation mode
   END_VAR

   VAR_TEMP 
      TIMER_ON : Bool;   // Timer signal ON
      TIMER_OFF : Bool;   // Timer signal OFF
   END_VAR


BEGIN
	
	(*
	Network 1: Start up
	*)
	IF #RESTART= true THEN
	  #QON:= false;
	  #QON_DELAY:=false;
	  #QOFF:=true;
	  #QOFF_DELAY:=false;
	  #OPdwCmd:=0;
	END_IF;
	
	(*
	Network 2: Simulation On/Off
	Vaiable: OPdwCmd  Bit:  20  =  Process
	Vaiable: OPdwCmd  Bit:  21  =  Simulation
	*)
	IF (#LIOP_SEL=true AND #L_SIM=true) OR (#OPdwCmd.%X21=true AND #LIOP_SEL=false) THEN
	  #QSIM:=true;
	  #OPdwCmd.%X20:=false;
	  #OPdwCmd.%X21:=false;
	ELSIF (#LIOP_SEL=true AND #L_SIM=false) OR (#OPdwCmd.%X20=true AND #LIOP_SEL=false) THEN
	  #QSIM:= false;
	  #OPdwCmd.%X20:=false;
	  #OPdwCmd.%X21:=false;
	END_IF;
	
	(*
	Network 3: Reset Operation
	Vaiable: OPdwCmd  Bit:  24  =  Reset
	*)
	// Rising edge by linking
	IF #L_RESET=true AND #SE_L_RESET_LINK_COND=false THEN
	  #SE_L_RESET_LINK:=true;
	  #SE_L_RESET_LINK_COND:=true;
	ELSIF #L_RESET=true AND #SE_L_RESET_LINK_COND=true THEN
	  #SE_L_RESET_LINK:=false;
	ELSE
	  #SE_L_RESET_LINK_COND:=false;
	END_IF;
	// Rising edge by operator
	IF #OPdwCmd.%X24=true THEN
	  #SE_L_RESET_OP:=true;
	  #OPdwCmd.%X24:=false;
	ELSE
	  #SE_L_RESET_OP:=false;
	END_IF;
	// Reset error
	// #OP_RESET:=(#LIOP_SEL AND #SE_L_RESET_LINK) OR (#SE_L_RESET_OP AND NOT #LIOP_SEL);
	#OP_RESET := (#SE_L_RESET_LINK OR (#SE_L_RESET_OP AND NOT #LIOP_SEL)) AND NOT #LOCK;
	
	(*
	Network 4: Create input signal
	*)
	#QINP:=#INP XOR #INP_NEG;
	
	(*
	Network 6: Check errors
	*)
	#QERR_EXTERN:=#ERR_EXTERN;
	// Check for interlock
	IF #LOCK=true AND (#QON=true OR #QON_DELAY=true OR #QOFF_DELAY=true) THEN
	  #QLOCK:=true;
	ELSIF #OP_RESET=true THEN
	  #QLOCK:=false;
	END_IF;
	// Check for general error
	IF #QERR_EXTERN=true OR #QLOCK=true THEN
	  #QERR:=true;
	ELSIF #OP_RESET=true THEN
	  #QERR:=false;
	END_IF;
	
	(*
	Network 7: TOGGLE Simulation Bit
	*)
	IF #OPdwCmd.%X4=true AND #QSIM=true THEN
	  #SINP_SIM := NOT #SINP_SIM;
	  #OPdwCmd.%X4:=false;
	END_IF;
	
	(*
	Network 8: Bumpless switch to simulation mode
	*)
	IF #QSIM=false THEN
	    #INP_SIM := #QINP;  
	END_IF;
	
	(*
	Network 9: Evaluate for delays
	*)
	// Evaluate for ON delay
	IF #DELAY_TIME<> t#1ms THEN
	  #DELAY_ON:=true;
	ELSE
	  #DELAY_ON:=false; 
	END_IF;
	// Evaluate for OFF delay
	IF #DELAY_TIME_OFF <> t#1ms THEN
	  #DELAY_OFF:=true;
	ELSE
	  #DELAY_OFF:=false;
	END_IF;
	
	(*
	Network 10: Settting ON/OFF
	*)
	// Delay time for setting on
	    #T_ON(IN:=#DELAY_ON AND #QON_DELAY,
	           PT:=#DELAY_TIME,
	           Q=>#TIMER_ON,
	           ET=>#QDELAY_TIME);
	// Delay time for setting off               
	    #T_OFF(IN:=#DELAY_OFF AND #QOFF_DELAY ,
	            PT:=#DELAY_TIME_OFF,
	            Q=>#TIMER_OFF,
	            ET=>#QDELAY_TIME_OFF);
	
	IF #QERR=false AND #LOCK=false THEN
	  // Sets variable, for closing process in progress
	  #QON_DELAY:=((NOT #QSIM AND #QINP) OR (#QSIM AND (#INP_SIM OR #SINP_SIM)))AND NOT #QON;
	  // Sets variable, for opening process in progress
	  #QOFF_DELAY:=((NOT #QSIM AND NOT #QINP) OR (#QSIM AND NOT (#INP_SIM OR #SINP_SIM)))AND NOT #QOFF;
	
	  // Sets variable, for ON/OFF   
	  IF #TIMER_ON=true OR (#QINP=true AND #DELAY_ON=false) OR (#OLD_SIG_COND=true AND #QOFF_DELAY=false) THEN
	    // On case
	     #QON:=true;
	     #QOFF:=false;
	     #OLD_SIG_COND:=true;
	   ELSIF #TIMER_OFF=true OR (#QINP=false AND #DELAY_OFF=false) OR (#OLD_SIG_COND=false AND #QON_DELAY=false) THEN
	     // Off case
	     #QON:=false;
	     #QOFF:=true;
	     #OLD_SIG_COND:=false;
	   ELSE
	     // switch ON <--> OFF case
	     #QON:=false;
	     #QOFF:=false;
	   END_IF;
	ELSE
	   // Error case
	     #QON_DELAY:=false;
	     #QOFF_DELAY:=false;
	     #QON:=false;
	     #QOFF:=NOT #QERR;
	     #OLD_SIG_COND:=false;
	END_IF;
	
	(*
	Network 11: QOUT
	*)
	#QOUT := #QON OR #QOFF_DELAY;
	
	(*
	Network 12: Influence visibility of faceplate window
	*)
	IF #OP_VISIBILITY<>#VISIBILITY_OLD THEN
	  #VISIBILITY_OLD:=#OP_VISIBILITY;
	  #VISIBILITY:=#OP_VISIBILITY;
	ELSIF #VISIBILITY<>#VISIBILITY_OLD THEN
	  #VISIBILITY_OLD:=#VISIBILITY;
	  #OP_VISIBILITY:=#VISIBILITY;
	END_IF;
	
	(*
	Network 13: Set state for HMI
	*)
	#QdwState.%X0:=#QOFF;
	#QdwState.%X1:=#QOFF_DELAY;
	#QdwState.%X2:=#QON;
	#QdwState.%X3:=#QON_DELAY;
	#QdwState.%X4:=false;
	#QdwState.%X5:=false;
	#QdwState.%X6:=false;
	#QdwState.%X7:=false;
	#QdwState.%X8:=#QINP;
	#QdwState.%X9:=false;
	#QdwState.%X10:=false;
	#QdwState.%X11:=false;
	#QdwState.%X12:=#INP_NEG;
	#QdwState.%X13:=#SINP_SIM;
	#QdwState.%X14:=false;
	#QdwState.%X15:=false;
	#QdwState.%X16:=false;
	#QdwState.%X17:=false;
	#QdwState.%X18:=#QSIM;
	#QdwState.%X19:=false;
	#QdwState.%X20:=false;
	#QdwState.%X21:=false;
	#QdwState.%X22:=false;
	#QdwState.%X23:=false;
	#QdwState.%X24:=#QERR;
	#QdwState.%X25:=#QERR_EXTERN;
	#QdwState.%X26:=#QLOCK;
	#QdwState.%X27:=#LOCK;
	#QdwState.%X28:=false;
	#QdwState.%X29:=false;
	#QdwState.%X30:=false;
	#QdwState.%X31:=false;
	
	(*
	Network 14: Bit alarm procedure
	*)
	#QwAlarm.%X0:=false;
	#QwAlarm.%X1:=false;
	#QwAlarm.%X2:=false;
	#QwAlarm.%X3:=false;
	#QwAlarm.%X4:=#QLOCK;
	#QwAlarm.%X5:=false;
	#QwAlarm.%X6:=#QERR_EXTERN;
	#QwAlarm.%X7:=#QERR;
	#QwAlarm.%X8:=#QON;
	#QwAlarm.%X9:=#QON_DELAY;
	#QwAlarm.%X10:=false;
	#QwAlarm.%X11:=false;
	#QwAlarm.%X12:=#LOCK;
	#QwAlarm.%X13:=false;
	#QwAlarm.%X14:=false;
	#QwAlarm.%X15:=#QSIM;
END_FUNCTION_BLOCK

FUNCTION_BLOCK "BFT_ChiliAwetan"   // FB361, LAD
{ S7_Optimized_Access := 'TRUE' }
VERSION : 0.1
// stored: AutoNumber false, IsIECCheckEnabled false, IsRetainMemResEnabled false, MemoryReserve 100, SetENOAutomatically false, UDAEnableTagReadback false
   VAR_INPUT
      IN_FBAV_Inload : Bool;
      IN_FBAV_Outlet : Bool;
      IN_FBAV_Transfer : Bool;
      IN_FBAV_CIP_Tank : Bool;
      IN_FBAV_CIP_Line : Bool;
      IN_FBP_Inload : Bool;
      IN_FBP_Inload_SP : Real;
      IN_FBP_Transfer : Bool;
      IN_FBP_Transfer_SP : Real;
      IN_FBP_CIP : Bool;
      IN_FBP_CIP_Sp : Real;
      IN_LT01 : Real;
      "LCS Start" : Bool;
      "LCS Stop" : Bool;
      "LCS EMS" : Bool;
      IN_Dose_Run : Bool;
      IN_Dose_Held : Bool;
      IN_Dose_Complete : Bool;
      IN_Dose_Header_1 : Bool;
      IN_Dose_Header_2 : Bool;
      IN_Dose_Valve_Cmd : Bool;
      IN_Dose_Pump_Cmd : Bool;
      IN_Dose_Pump_Sp : Real;
      IN_Dose_LineOK : Bool;
      "Inload Busy" : Bool;
      IN_Prod_Ready : Bool;
      IN_Prod_LineOpen : Bool;
      IN_SupplyOn : Bool;
      IN_Prod_Transfer_Comp : Bool;
      "CIP Pulse" : Bool;
      "CIP Supply ON" : Bool;
      "CIP Req OK" : Bool;
      "CIP Complete" : Bool;
      "CIP Busy" : Bool;
   END_VAR
   VAR_OUTPUT
      Out_AV_Inload : Bool;
      Out_AV_Outlet : Bool;
      Out_AV_Transfer : Bool;
      Out_AV_CIP_Tank : Bool;
      Out_AV_CIP_Line : Bool;
      Out_P_Inload : Bool;
      Out_P_Inload_Sp : Real;
      Out_P_Transfer : Bool;
      Out_P_Transfer_Sp : Real;
      Out_P_CIP : Bool;
      Out_P_CIP_Sp : Real;
      Out_Prod_Req : Bool;
      Out_Prod_LineOpen : Bool;
      Out_CIP_Req : Bool;
      Out_CIP_LineOpen : Bool;
   END_VAR
   VAR
      Cmd : Struct
         Inload : Bool;
         Ready_for_Tranfer : Bool;
         CIP_Tank : Bool;
         CIP_Line : Bool;
      END_STRUCT;
   END_VAR
   VAR RETAIN
      Param : Struct
         SP_Level_LL : Real := 10.0;
         SP_Level_ML : Real := 80.0;
         SP_Level_HL : Real := 100.0;
         SupplyPump_SP_Speed : Real := 80.0;
         L_Hi_Lim : Real := 100.0;
         L_Lo_Lim : Real := 0.0;
         L_Hys : Real := 2.0;
         FlushingTime : DInt := 10000;
         CIP_Trf_SP_Speed : Real := 80.0;
         CIP_Ret_ON_SP : Real := 5.0;
         CIP_Ret_OFF_SP : Real;
      END_STRUCT;
   END_VAR
   VAR
      State : Struct   // Tank in loading state
         Tank_LL : Bool;
         Tank_ML : Bool;
         Tank_HL : Bool;
         Tank_inCIP : Bool;
         Tank_CIP_Enable : Bool;
         Line_inCIP : Bool;
         Line_CIP_Enable : Bool;
         CIP_Return_On : Bool;
         Inloading : Bool;
         Inload_Enable : Bool;
         Ready_For_Transfer : Bool;
         Ready_For_Transfer_Ena : Bool;
         Tank_Available : Bool;
         Transfer_On_Prog : Bool;
      END_STRUCT;
      alwaysON : Bool;
      L_Hys_Abs : Real;
      Hys_Level_HL : Real;
      Hys_Level_ML : Real;
      Hys_Level_LL : Real;
      r : Struct
         PosE1 : Bool;
         PosE2 : Bool;
         PosE3 : Bool;
         PosE4 : Bool;
         PosE5 : Bool;
         PosE6 : Bool;
         PosE7 : Bool;
         PosE8 : Bool;
         PosE9 : Bool;
         PosE10 : Bool;
         PosE11 : Bool;
         PosE12 : Bool;
         PosE13 : Bool;
         PosE14 : Bool;
         PosE15 : Bool;
         PosE16 : Bool;
         PosE17 : Bool;
         PosE18 : Bool;
         PosE19 : Bool;
         PosE20 : Bool;
         PosE21 : Bool;
         PosE22 : Bool;
         PosE23 : Bool;
         PosE24 : Bool;
         PosE25 : Bool;
         PosE26 : Bool;
         PosE27 : Bool;
         PosE28 : Bool;
         PosE29 : Bool;
         PosE30 : Bool;
         PosE31 : Bool;
         PosE32 : Bool;
      END_STRUCT;
      Actuator : Struct
         AV_Inload : Bool;
         AV_Outlet : Bool;
         AV_Transfer : Bool;
         AV_CIP_Tank : Bool;
         AV_CIP_Line : Bool;
         P_Transfer : Bool;
         P_Inload : Bool;
         P_CIP : Bool;
      END_STRUCT;
      FlushingTim : TON_TIME;
      SPumpTim { S7_SetPoint := 'True'} : TON_TIME;
      AVinloadTim { S7_SetPoint := 'True'} : TON_TIME;
      Pump_TF_On_Time { S7_SetPoint := 'True'} : TON_TIME;
   END_VAR
   VAR_TEMP   // added for the SCL form of the ladder/FBD networks
      _w1 : Bool;
      _w2 : Bool;
   END_VAR
BEGIN

REGION Network 1: Always_ON
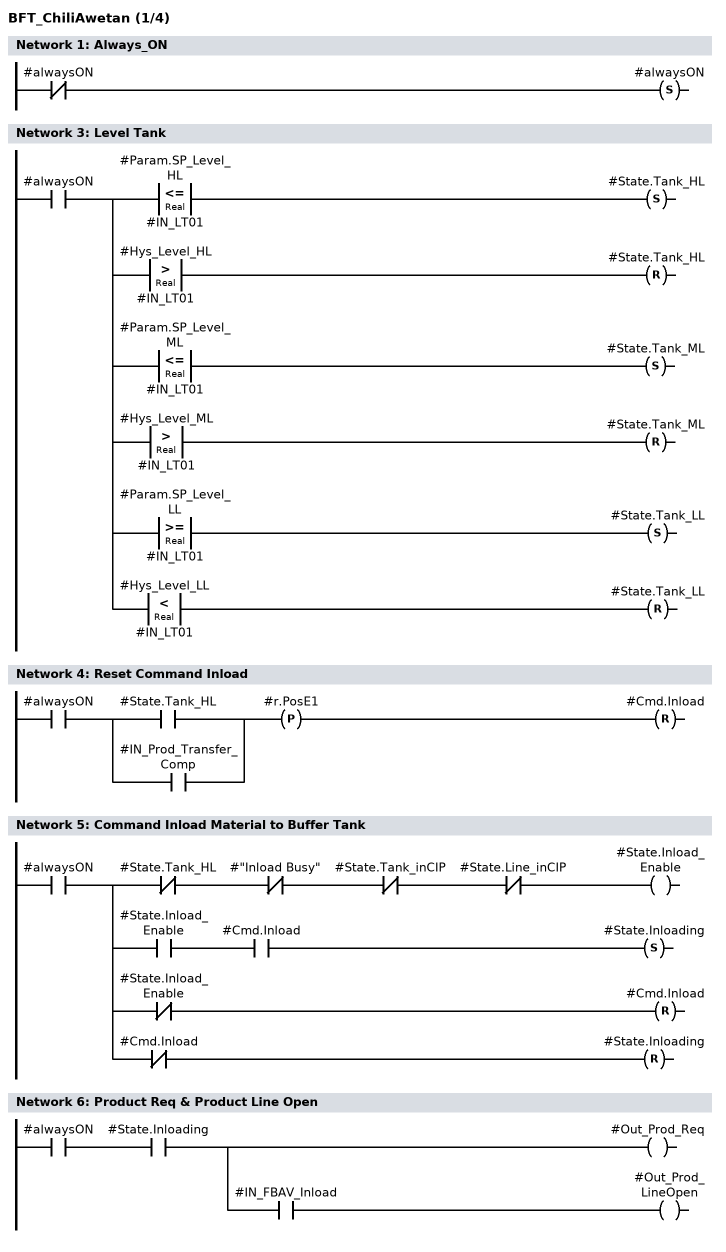
   RUNG wire#powerrail
      I_Contact( #alwaysON )
      S_Coil( #alwaysON )
   END_RUNG
   // the same network as SCL:
   IF NOT #alwaysON THEN #alwaysON := TRUE; END_IF;
END_REGION

NETWORK
TITLE = Hys Calculation
//Level Hys Absolute
      L     #Param.L_Hi_Lim;
      L     #Param.L_Lo_Lim;
      -R;
      L     100.0;
      /R;
      L     #Param.L_Hys;
      *R;
      T     #L_Hys_Abs;
//Tank High Level
      L     #Param.SP_Level_HL;
      L     #L_Hys_Abs;
      -R;
      T     #Hys_Level_HL;
//Tank Mid Level
      L     #Param.SP_Level_ML;
      L     #L_Hys_Abs;
      -R;
      T     #Hys_Level_ML;
//Tank Low Level
      L     #Param.SP_Level_LL;
      L     #L_Hys_Abs;
      +R;
      T     #Hys_Level_LL;


REGION Network 3: Level Tank
   RUNG wire#powerrail
      Contact( #alwaysON )
      wire#w1
      { S7_Templates := "SrcType := Real" } LE_Contact(in1 := #Param.SP_Level_HL, in2 := #IN_LT01)
      S_Coil( #State.Tank_HL )
   END_RUNG
   RUNG wire#w1
      { S7_Templates := "SrcType := Real" } GT_Contact(in1 := #Hys_Level_HL, in2 := #IN_LT01)
      R_Coil( #State.Tank_HL )
   END_RUNG
   RUNG wire#w1
      { S7_Templates := "SrcType := Real" } LE_Contact(in1 := #Param.SP_Level_ML, in2 := #IN_LT01)
      S_Coil( #State.Tank_ML )
   END_RUNG
   RUNG wire#w1
      { S7_Templates := "SrcType := Real" } GT_Contact(in1 := #Hys_Level_ML, in2 := #IN_LT01)
      R_Coil( #State.Tank_ML )
   END_RUNG
   RUNG wire#w1
      { S7_Templates := "SrcType := Real" } GE_Contact(in1 := #Param.SP_Level_LL, in2 := #IN_LT01)
      S_Coil( #State.Tank_LL )
   END_RUNG
   RUNG wire#w1
      { S7_Templates := "SrcType := Real" } LT_Contact(in1 := #Hys_Level_LL, in2 := #IN_LT01)
      R_Coil( #State.Tank_LL )
   END_RUNG
   // the same network as SCL:
   IF #alwaysON AND (#Param.SP_Level_HL <= #IN_LT01) THEN #State.Tank_HL := TRUE; END_IF;
   IF #alwaysON AND (#Hys_Level_HL > #IN_LT01) THEN #State.Tank_HL := FALSE; END_IF;
   IF #alwaysON AND (#Param.SP_Level_ML <= #IN_LT01) THEN #State.Tank_ML := TRUE; END_IF;
   IF #alwaysON AND (#Hys_Level_ML > #IN_LT01) THEN #State.Tank_ML := FALSE; END_IF;
   IF #alwaysON AND (#Param.SP_Level_LL >= #IN_LT01) THEN #State.Tank_LL := TRUE; END_IF;
   IF #alwaysON AND (#Hys_Level_LL < #IN_LT01) THEN #State.Tank_LL := FALSE; END_IF;
END_REGION

REGION Network 4: Reset Command Inload
   RUNG wire#powerrail
      Contact( #alwaysON )
      wire#w1
      Contact( #State.Tank_HL )
      wire#w2
      P_Trig( #r.PosE1 )
      R_Coil( #Cmd.Inload )
   END_RUNG
   RUNG wire#w1
      Contact( #IN_Prod_Transfer_Comp )
   END_RUNG wire#w2
   // the same network as SCL:
   #_w1 := #alwaysON AND (#State.Tank_HL OR #IN_Prod_Transfer_Comp);
   #_w2 := #_w1 AND NOT #r.PosE1;   // rising edge
   #r.PosE1 := #_w1;
   IF #_w2 THEN #Cmd.Inload := FALSE; END_IF;
END_REGION

REGION Network 5: Command Inload Material to Buffer Tank
   RUNG wire#powerrail
      Contact( #alwaysON )
      wire#w1
      I_Contact( #State.Tank_HL )
      I_Contact( #"Inload Busy" )
      I_Contact( #State.Tank_inCIP )
      I_Contact( #State.Line_inCIP )
      Coil( #State.Inload_Enable )
   END_RUNG
   RUNG wire#w1
      Contact( #State.Inload_Enable )
      Contact( #Cmd.Inload )
      S_Coil( #State.Inloading )
   END_RUNG
   RUNG wire#w1
      I_Contact( #State.Inload_Enable )
      R_Coil( #Cmd.Inload )
   END_RUNG
   RUNG wire#w1
      I_Contact( #Cmd.Inload )
      R_Coil( #State.Inloading )
   END_RUNG
   // the same network as SCL:
   #State.Inload_Enable := #alwaysON AND NOT #State.Tank_HL AND NOT #"Inload Busy" AND NOT #State.Tank_inCIP AND NOT #State.Line_inCIP;
   IF #alwaysON AND #State.Inload_Enable AND #Cmd.Inload THEN #State.Inloading := TRUE; END_IF;
   IF #alwaysON AND NOT #State.Inload_Enable THEN #Cmd.Inload := FALSE; END_IF;
   IF #alwaysON AND NOT #Cmd.Inload THEN #State.Inloading := FALSE; END_IF;
END_REGION

REGION Network 6: Product Req & Product Line Open
   RUNG wire#powerrail
      Contact( #alwaysON )
      Contact( #State.Inloading )
      wire#w1
      Coil( #Out_Prod_Req )
   END_RUNG
   RUNG wire#w1
      Contact( #IN_FBAV_Inload )
      Coil( #Out_Prod_LineOpen )
   END_RUNG
   // the same network as SCL:
   #Out_Prod_Req := #alwaysON AND #State.Inloading;
   #Out_Prod_LineOpen := #Out_Prod_Req AND #IN_FBAV_Inload;
END_REGION

REGION Network 8: Tank Ready for Transfer to Blending
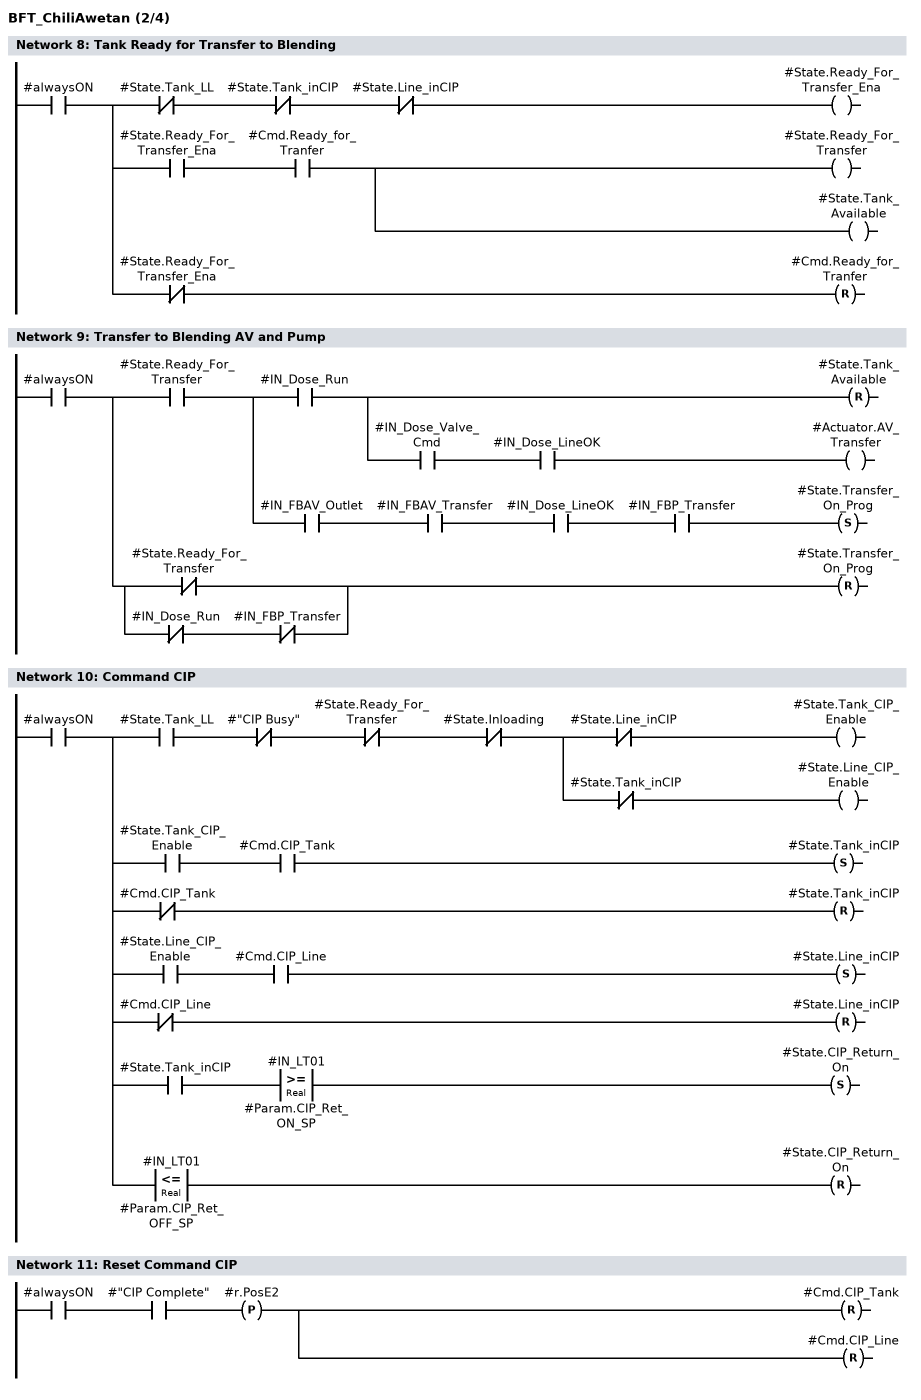
   RUNG wire#powerrail
      Contact( #alwaysON )
      wire#w1
      I_Contact( #State.Tank_LL )
      I_Contact( #State.Tank_inCIP )
      I_Contact( #State.Line_inCIP )
      Coil( #State.Ready_For_Transfer_Ena )
   END_RUNG
   RUNG wire#w1
      Contact( #State.Ready_For_Transfer_Ena )
      Contact( #Cmd.Ready_for_Tranfer )
      wire#w2
      Coil( #State.Ready_For_Transfer )
   END_RUNG
   RUNG wire#w2
      Coil( #State.Tank_Available )
   END_RUNG
   RUNG wire#w1
      I_Contact( #State.Ready_For_Transfer_Ena )
      R_Coil( #Cmd.Ready_for_Tranfer )
   END_RUNG
   // the same network as SCL:
   #State.Ready_For_Transfer_Ena := #alwaysON AND NOT #State.Tank_LL AND NOT #State.Tank_inCIP AND NOT #State.Line_inCIP;
   #State.Ready_For_Transfer := #alwaysON AND #State.Ready_For_Transfer_Ena AND #Cmd.Ready_for_Tranfer;
   #State.Tank_Available := #State.Ready_For_Transfer;
   IF #alwaysON AND NOT #State.Ready_For_Transfer_Ena THEN #Cmd.Ready_for_Tranfer := FALSE; END_IF;
END_REGION

REGION Network 9: Transfer to Blending AV and Pump
   RUNG wire#powerrail
      Contact( #alwaysON )
      wire#w1
      Contact( #State.Ready_For_Transfer )
      wire#w2
      Contact( #IN_Dose_Run )
      wire#w3
      R_Coil( #State.Tank_Available )
   END_RUNG
   RUNG wire#w3
      Contact( #IN_Dose_Valve_Cmd )
      Contact( #IN_Dose_LineOK )
      Coil( #Actuator.AV_Transfer )
   END_RUNG
   RUNG wire#w2
      Contact( #IN_FBAV_Outlet )
      Contact( #IN_FBAV_Transfer )
      Contact( #IN_Dose_LineOK )
      Contact( #IN_FBP_Transfer )
      S_Coil( #State.Transfer_On_Prog )
   END_RUNG
   RUNG wire#w1
      I_Contact( #State.Ready_For_Transfer )
      wire#w4
      R_Coil( #State.Transfer_On_Prog )
   END_RUNG
   RUNG wire#w1
      I_Contact( #IN_Dose_Run )
      I_Contact( #IN_FBP_Transfer )
   END_RUNG wire#w4
   // the same network as SCL:
   #_w1 := #alwaysON AND #State.Ready_For_Transfer;
   #_w2 := #_w1 AND #IN_Dose_Run;
   IF #_w2 THEN #State.Tank_Available := FALSE; END_IF;
   #Actuator.AV_Transfer := #_w2 AND #IN_Dose_Valve_Cmd AND #IN_Dose_LineOK;
   IF #_w1 AND #IN_FBAV_Outlet AND #IN_FBAV_Transfer AND #IN_Dose_LineOK AND #IN_FBP_Transfer THEN
       #State.Transfer_On_Prog := TRUE;
   END_IF;
   IF #alwaysON AND (NOT #State.Ready_For_Transfer OR (NOT #IN_Dose_Run AND NOT #IN_FBP_Transfer)) THEN
       #State.Transfer_On_Prog := FALSE;
   END_IF;
END_REGION

REGION Network 10: Command CIP
   RUNG wire#powerrail
      Contact( #alwaysON )
      wire#w1
      Contact( #State.Tank_LL )
      I_Contact( #"CIP Busy" )
      I_Contact( #State.Ready_For_Transfer )
      I_Contact( #State.Inloading )
      wire#w2
      I_Contact( #State.Line_inCIP )
      Coil( #State.Tank_CIP_Enable )
   END_RUNG
   RUNG wire#w2
      I_Contact( #State.Tank_inCIP )
      Coil( #State.Line_CIP_Enable )
   END_RUNG
   RUNG wire#w1
      Contact( #State.Tank_CIP_Enable )
      Contact( #Cmd.CIP_Tank )
      S_Coil( #State.Tank_inCIP )
   END_RUNG
   RUNG wire#w1
      I_Contact( #Cmd.CIP_Tank )
      R_Coil( #State.Tank_inCIP )
   END_RUNG
   RUNG wire#w1
      Contact( #State.Line_CIP_Enable )
      Contact( #Cmd.CIP_Line )
      S_Coil( #State.Line_inCIP )
   END_RUNG
   RUNG wire#w1
      I_Contact( #Cmd.CIP_Line )
      R_Coil( #State.Line_inCIP )
   END_RUNG
   RUNG wire#w1
      Contact( #State.Tank_inCIP )
      { S7_Templates := "SrcType := Real" } GE_Contact(in1 := #IN_LT01, in2 := #Param.CIP_Ret_ON_SP)
      S_Coil( #State.CIP_Return_On )
   END_RUNG
   RUNG wire#w1
      { S7_Templates := "SrcType := Real" } LE_Contact(in1 := #IN_LT01, in2 := #Param.CIP_Ret_OFF_SP)
      R_Coil( #State.CIP_Return_On )
   END_RUNG
   // the same network as SCL:
   #_w1 := #alwaysON AND #State.Tank_LL AND NOT #"CIP Busy" AND NOT #State.Ready_For_Transfer AND NOT #State.Inloading;
   #State.Tank_CIP_Enable := #_w1 AND NOT #State.Line_inCIP;
   #State.Line_CIP_Enable := #_w1 AND NOT #State.Tank_inCIP;
   IF #alwaysON AND #State.Tank_CIP_Enable AND #Cmd.CIP_Tank THEN #State.Tank_inCIP := TRUE; END_IF;
   IF #alwaysON AND NOT #Cmd.CIP_Tank THEN #State.Tank_inCIP := FALSE; END_IF;
   IF #alwaysON AND #State.Line_CIP_Enable AND #Cmd.CIP_Line THEN #State.Line_inCIP := TRUE; END_IF;
   IF #alwaysON AND NOT #Cmd.CIP_Line THEN #State.Line_inCIP := FALSE; END_IF;
   IF #alwaysON AND #State.Tank_inCIP AND (#IN_LT01 >= #Param.CIP_Ret_ON_SP) THEN
       #State.CIP_Return_On := TRUE;
   END_IF;
   IF #alwaysON AND (#IN_LT01 <= #Param.CIP_Ret_OFF_SP) THEN #State.CIP_Return_On := FALSE; END_IF;
END_REGION

REGION Network 11: Reset Command CIP
   RUNG wire#powerrail
      Contact( #alwaysON )
      Contact( #"CIP Complete" )
      P_Trig( #r.PosE2 )
      wire#w1
      R_Coil( #Cmd.CIP_Tank )
   END_RUNG
   RUNG wire#w1
      R_Coil( #Cmd.CIP_Line )
   END_RUNG
   // the same network as SCL:
   #_w1 := #alwaysON AND #"CIP Complete";
   #_w2 := #_w1 AND NOT #r.PosE2;   // rising edge
   #r.PosE2 := #_w1;
   IF #_w2 THEN
       #Cmd.CIP_Tank := FALSE;
       #Cmd.CIP_Line := FALSE;
   END_IF;
END_REGION

REGION Network 12: CIP Request and CIP Line Open
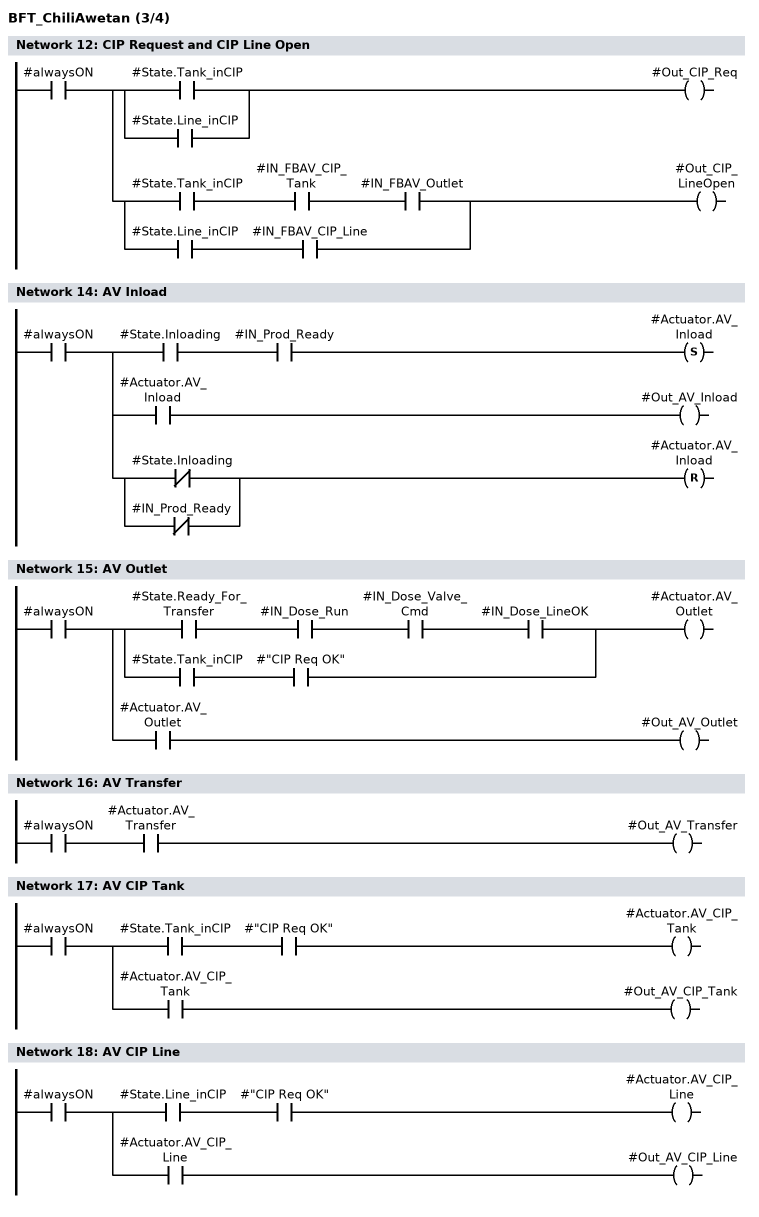
   RUNG wire#powerrail
      Contact( #alwaysON )
      wire#w1
      Contact( #State.Tank_inCIP )
      wire#w2
      Coil( #Out_CIP_Req )
   END_RUNG
   RUNG wire#w1
      Contact( #State.Line_inCIP )
   END_RUNG wire#w2
   RUNG wire#w1
      Contact( #State.Tank_inCIP )
      Contact( #IN_FBAV_CIP_Tank )
      Contact( #IN_FBAV_Outlet )
      wire#w3
      Coil( #Out_CIP_LineOpen )
   END_RUNG
   RUNG wire#w1
      Contact( #State.Line_inCIP )
      Contact( #IN_FBAV_CIP_Line )
   END_RUNG wire#w3
   // the same network as SCL:
   #Out_CIP_Req := #alwaysON AND (#State.Tank_inCIP OR #State.Line_inCIP);
   #Out_CIP_LineOpen := #alwaysON AND ((#State.Tank_inCIP AND #IN_FBAV_CIP_Tank AND #IN_FBAV_Outlet) OR (#State.Line_inCIP AND #IN_FBAV_CIP_Line));
END_REGION

REGION Network 14: AV Inload
   RUNG wire#powerrail
      Contact( #alwaysON )
      wire#w1
      Contact( #State.Inloading )
      Contact( #IN_Prod_Ready )
      S_Coil( #Actuator.AV_Inload )
   END_RUNG
   RUNG wire#w1
      Contact( #Actuator.AV_Inload )
      Coil( #Out_AV_Inload )
   END_RUNG
   RUNG wire#w1
      I_Contact( #State.Inloading )
      wire#w2
      R_Coil( #Actuator.AV_Inload )
   END_RUNG
   RUNG wire#w1
      I_Contact( #IN_Prod_Ready )
   END_RUNG wire#w2
   // the same network as SCL:
   IF #alwaysON AND #State.Inloading AND #IN_Prod_Ready THEN #Actuator.AV_Inload := TRUE; END_IF;
   #Out_AV_Inload := #alwaysON AND #Actuator.AV_Inload;
   IF #alwaysON AND (NOT #State.Inloading OR NOT #IN_Prod_Ready) THEN #Actuator.AV_Inload := FALSE; END_IF;
END_REGION

REGION Network 15: AV Outlet
   RUNG wire#powerrail
      Contact( #alwaysON )
      wire#w1
      Contact( #State.Ready_For_Transfer )
      Contact( #IN_Dose_Run )
      Contact( #IN_Dose_Valve_Cmd )
      Contact( #IN_Dose_LineOK )
      wire#w2
      Coil( #Actuator.AV_Outlet )
   END_RUNG
   RUNG wire#w1
      Contact( #State.Tank_inCIP )
      Contact( #"CIP Req OK" )
   END_RUNG wire#w2
   RUNG wire#w1
      Contact( #Actuator.AV_Outlet )
      Coil( #Out_AV_Outlet )
   END_RUNG
   // the same network as SCL:
   #Actuator.AV_Outlet := #alwaysON AND ((#State.Ready_For_Transfer AND #IN_Dose_Run AND #IN_Dose_Valve_Cmd AND #IN_Dose_LineOK) OR (#State.Tank_inCIP AND #"CIP Req OK"));
   #Out_AV_Outlet := #alwaysON AND #Actuator.AV_Outlet;
END_REGION

REGION Network 16: AV Transfer
   RUNG wire#powerrail
      Contact( #alwaysON )
      Contact( #Actuator.AV_Transfer )
      Coil( #Out_AV_Transfer )
   END_RUNG
   // the same network as SCL:
   #Out_AV_Transfer := #alwaysON AND #Actuator.AV_Transfer;
END_REGION

REGION Network 17: AV CIP Tank
   RUNG wire#powerrail
      Contact( #alwaysON )
      wire#w1
      Contact( #State.Tank_inCIP )
      Contact( #"CIP Req OK" )
      Coil( #Actuator.AV_CIP_Tank )
   END_RUNG
   RUNG wire#w1
      Contact( #Actuator.AV_CIP_Tank )
      Coil( #Out_AV_CIP_Tank )
   END_RUNG
   // the same network as SCL:
   #Actuator.AV_CIP_Tank := #alwaysON AND #State.Tank_inCIP AND #"CIP Req OK";
   #Out_AV_CIP_Tank := #alwaysON AND #Actuator.AV_CIP_Tank;
END_REGION

REGION Network 18: AV CIP Line
   RUNG wire#powerrail
      Contact( #alwaysON )
      wire#w1
      Contact( #State.Line_inCIP )
      Contact( #"CIP Req OK" )
      Coil( #Actuator.AV_CIP_Line )
   END_RUNG
   RUNG wire#w1
      Contact( #Actuator.AV_CIP_Line )
      Coil( #Out_AV_CIP_Line )
   END_RUNG
   // the same network as SCL:
   #Actuator.AV_CIP_Line := #alwaysON AND #State.Line_inCIP AND #"CIP Req OK";
   #Out_AV_CIP_Line := #alwaysON AND #Actuator.AV_CIP_Line;
END_REGION

REGION Network 20: Pump Inload
